	{attribute 'TcIecLibraryType'}
	{attribute 'external_name' := 'F_VN_MultiplyImages_GUID_82AA580E_DA77_541C_61B6_148C085FBCB3'}
	(* Element-wise multiplication of two images using saturation arithmetics. *)
	FUNCTION F_VN_MultiplyImages : HRESULT
	VAR_INPUT
		ipSrcImage1	:	ITcVnImage;	(* First source image *)
		ipSrcImage2	:	ITcVnImage;	(* Second source image *)
		ipDestImage	:	REFERENCE TO ITcVnImage;	(* Destination image (An appropriate destination image will be created if required.) *)
		hrPrev	:	HRESULT;	(* HRESULT indicating the result of previous operations (If SUCCEEDED(hrPrev) equals false, no operation is executed.) *)
	END_VAR

END_FUNCTION

// Functions/Algebraic Image Operations/F_VN_MultiplyImageWithScalar

	{attribute 'TcIecLibraryType'}
	{attribute 'external_name' := 'F_VN_MultiplyImageWithScalar_GUID_B12B22BD_02D6_587A_7D30_3355393075B2'}
	(* Multiply each image pixel by a scalar value using saturation arithmetics. *)
	FUNCTION F_VN_MultiplyImageWithScalar : HRESULT
	VAR_INPUT
		fScalar	:	LREAL;	(* Scalar value *)
		ipSrcImage	:	ITcVnImage;	(* Source image *)
		ipDestImage	:	REFERENCE TO ITcVnImage;	(* Destination image (An appropriate destination image will be created if required.) *)
		hrPrev	:	HRESULT;	(* HRESULT indicating the result of previous operations (If SUCCEEDED(hrPrev) equals false, no operation is executed.) *)
	END_VAR

END_FUNCTION

// Functions/Algebraic Image Operations/F_VN_MultiplyImageWithVector

	{attribute 'TcIecLibraryType'}
	{attribute 'external_name' := 'F_VN_MultiplyImageWithVector_GUID_5A56ACBB_6C80_5F28_4A45_B28BE648BFEA'}
	(* Multiply each image pixel by a vector (1 element for each image channel) using saturation arithmetics. *)
	FUNCTION F_VN_MultiplyImageWithVector : HRESULT
	VAR_INPUT
		aVector	:	REFERENCE TO TcVnVector4_LREAL;	(* 4-element vector (1 element for each image channel. If the image has less channels, the further vector elements are ignored.) *)
		ipSrcImage	:	ITcVnImage;	(* Source image *)
		ipDestImage	:	REFERENCE TO ITcVnImage;	(* Destination image (An appropriate destination image will be created if required.) *)
		hrPrev	:	HRESULT;	(* HRESULT indicating the result of previous operations (If SUCCEEDED(hrPrev) equals false, no operation is executed.) *)
	END_VAR

END_FUNCTION

// Functions/Algebraic Image Operations/F_VN_SubtractImageFromScalar

	{attribute 'TcIecLibraryType'}
	{attribute 'external_name' := 'F_VN_SubtractImageFromScalar_GUID_B8AA2245_74B9_5AC2_4E76_135813C299C9'}
	(* Subtract each image pixel from a scalar value using saturation arithmetics. *)
	FUNCTION F_VN_SubtractImageFromScalar : HRESULT
	VAR_INPUT
		fScalar	:	LREAL;	(* Scalar value *)
		ipSrcImage	:	ITcVnImage;	(* Source image *)
		ipDestImage	:	REFERENCE TO ITcVnImage;	(* Destination image (An appropriate destination image will be created if required.) *)
		hrPrev	:	HRESULT;	(* HRESULT indicating the result of previous operations (If SUCCEEDED(hrPrev) equals false, no operation is executed.) *)
	END_VAR

END_FUNCTION

// Functions/Algebraic Image Operations/F_VN_SubtractImageFromVector

	{attribute 'TcIecLibraryType'}
	{attribute 'external_name' := 'F_VN_SubtractImageFromVector_GUID_17517F7A_96FF_563D_5F02_C474E2D7CC0C'}
	(* Subtract each image pixel from a vector (1 element for each image channel) using saturation arithmetics. *)
	FUNCTION F_VN_SubtractImageFromVector : HRESULT
	VAR_INPUT
		aVector	:	REFERENCE TO TcVnVector4_LREAL;	(* 4-element vector (1 element for each image channel. If the image has less channels, the further vector elements are ignored.) *)
		ipSrcImage	:	ITcVnImage;	(* Source image *)
		ipDestImage	:	REFERENCE TO ITcVnImage;	(* Destination image (An appropriate destination image will be created if required.) *)
		hrPrev	:	HRESULT;	(* HRESULT indicating the result of previous operations (If SUCCEEDED(hrPrev) equals false, no operation is executed.) *)
	END_VAR

END_FUNCTION

// Functions/Algebraic Image Operations/F_VN_SubtractImages

	{attribute 'TcIecLibraryType'}
	{attribute 'external_name' := 'F_VN_SubtractImages_GUID_93AB2995_6F42_52A0_4DD8_5441458B881F'}
	(* Element-wise subtraction of two images using saturation arithmetics. *)
	FUNCTION F_VN_SubtractImages : HRESULT
	VAR_INPUT
		ipSrcImage1	:	ITcVnImage;	(* First source image (minuend) *)
		ipSrcImage2	:	ITcVnImage;	(* Second source image (subtrahend) *)
		ipDestImage	:	REFERENCE TO ITcVnImage;	(* Destination image (An appropriate destination image will be created if required.) *)
		hrPrev	:	HRESULT;	(* HRESULT indicating the result of previous operations (If SUCCEEDED(hrPrev) equals false, no operation is executed.) *)
	END_VAR

END_FUNCTION

// Functions/Algebraic Image Operations/F_VN_SubtractScalarFromImage

	{attribute 'TcIecLibraryType'}
	{attribute 'external_name' := 'F_VN_SubtractScalarFromImage_GUID_4A75C512_59C5_5BEC_5299_C05E617DC6EB'}
	(* Subtract a scalar value from each image pixel using saturation arithmetics. *)
	FUNCTION F_VN_SubtractScalarFromImage : HRESULT
	VAR_INPUT
		ipSrcImage	:	ITcVnImage;	(* Source image *)
		fScalar	:	LREAL;	(* Scalar value *)
		ipDestImage	:	REFERENCE TO ITcVnImage;	(* Destination image (An appropriate destination image will be created if required.) *)
		hrPrev	:	HRESULT;	(* HRESULT indicating the result of previous operations (If SUCCEEDED(hrPrev) equals false, no operation is executed.) *)
	END_VAR

END_FUNCTION

// Functions/Algebraic Image Operations/F_VN_SubtractVectorFromImage

	{attribute 'TcIecLibraryType'}
	{attribute 'external_name' := 'F_VN_SubtractVectorFromImage_GUID_3A450D3E_E7EC_586B_54DB_8372F7AAF290'}
	(* Subtract a vector (1 element for each image channel) from each image pixel using saturation arithmetics. *)
	FUNCTION F_VN_SubtractVectorFromImage : HRESULT
	VAR_INPUT
		ipSrcImage	:	ITcVnImage;	(* Source image *)
		aVector	:	REFERENCE TO TcVnVector4_LREAL;	(* 4-element vector (1 element for each image channel. If the image has less channels, the further vector elements are ignored.) *)
		ipDestImage	:	REFERENCE TO ITcVnImage;	(* Destination image (An appropriate destination image will be created if required.) *)
		hrPrev	:	HRESULT;	(* HRESULT indicating the result of previous operations (If SUCCEEDED(hrPrev) equals false, no operation is executed.) *)
	END_VAR

END_FUNCTION

// Functions/Image Analysis/F_VN_CannyEdgeDetection

	{attribute 'TcIecLibraryType'}
	{attribute 'external_name' := 'F_VN_CannyEdgeDetection_GUID_AD5174D6_E5E1_5D48_5694_BB03C2CA2FDE'}
	(* Find edges using the Canny edge detection algorithm. *)
	FUNCTION F_VN_CannyEdgeDetection : HRESULT
	VAR_INPUT
		ipSrcImage	:	ITcVnImage;	(* Source image (elements of type USINT) *)
		ipDestImage	:	REFERENCE TO ITcVnImage;	(* Destination image (elements of type USINT. An appropriate destination image will be created if required.) *)
		fThresholdLow	:	LREAL;	(* Low threshold *)
		fThresholdHigh	:	LREAL;	(* High threshold *)
		hrPrev	:	HRESULT;	(* HRESULT indicating the result of previous operations (If SUCCEEDED(hrPrev) equals false, no operation is executed.) *)
	END_VAR

END_FUNCTION

// Functions/Image Analysis/F_VN_CannyEdgeDetectionExp

	{attribute 'TcIecLibraryType'}
	{attribute 'external_name' := 'F_VN_CannyEdgeDetectionExp_GUID_6D08A1F4_144F_582E_608D_60E37CF3A2B0'}
	(* Find edges using the Canny edge detection algorithm. (expert function) *)
	FUNCTION F_VN_CannyEdgeDetectionExp : HRESULT
	VAR_INPUT
		ipSrcImage	:	ITcVnImage;	(* Source image (elements of type USINT) *)
		ipDestImage	:	REFERENCE TO ITcVnImage;	(* Destination image (elements of type USINT. An appropriate destination image will be created if required.) *)
		fThresholdLow	:	LREAL;	(* Low threshold *)
		fThresholdHigh	:	LREAL;	(* High threshold *)
		nApertureSize	:	UDINT;	(* Aperture size for the Sobel operator (3, 5, 7) *)
		bL2Gradient	:	BOOL;	(* If true, the more accurate (and slower) L2 norm is used instead of the L1 norm *)
		hrPrev	:	HRESULT;	(* HRESULT indicating the result of previous operations (If SUCCEEDED(hrPrev) equals false, no operation is executed.) *)
	END_VAR

END_FUNCTION

// Functions/Image Analysis/F_VN_CountNonZeroPixels

	{attribute 'TcIecLibraryType'}
	{attribute 'external_name' := 'F_VN_CountNonZeroPixels_GUID_9D27D17F_B34D_59A9_5A50_23FA7CA7A721'}
	(* Counts the non-zero pixels in a single-channel image (e.g. useful to analyze threshold results). *)
	FUNCTION F_VN_CountNonZeroPixels : HRESULT
	VAR_INPUT
		ipSrcImage	:	ITcVnImage;	(* Source image (1 channel) *)
		nNonZero	:	REFERENCE TO ULINT;	(* Returns the number of non-zero pixels in ipSrcImage *)
		hrPrev	:	HRESULT;	(* HRESULT indicating the result of previous operations (If SUCCEEDED(hrPrev) equals false, no operation is executed.) *)
	END_VAR

END_FUNCTION

// Functions/Image Analysis/F_VN_DistanceTransformation

	{attribute 'TcIecLibraryType'}
	{attribute 'external_name' := 'F_VN_DistanceTransformation_GUID_4E9A92BB_223F_5813_612F_9AC3CDD271BA'}
	(* Calculates the distance transformation, which is the distance to the closest zero pixel in a binary image. *)
	FUNCTION F_VN_DistanceTransformation : HRESULT
	VAR_INPUT
		ipSrcImage	:	ITcVnImage;	(* Source image (USINT, 1 channel) *)
		ipDestImage	:	REFERENCE TO ITcVnImage;	(* Destination image (REAL, 1 channel. An appropriate destination image will be created if required.) *)
		eDistanceType	:	ETcVnDistanceType;	(* Distance computation method (supported: L1, L2, C) *)
		eMaskSize	:	ETcVnDistanceTransformationMask;	(* Size of the distance transformation mask *)
		hrPrev	:	HRESULT;	(* HRESULT indicating the result of previous operations (If SUCCEEDED(hrPrev) equals false, no operation is executed.) *)
	END_VAR

END_FUNCTION

// Functions/Image Analysis/F_VN_DistanceTransformationExp

	{attribute 'TcIecLibraryType'}
	{attribute 'external_name' := 'F_VN_DistanceTransformationExp_GUID_4CFD3356_1E5B_593C_50A2_5B385695B3A8'}
	(* Calculates the distance transformation, which is the distance to the closest zero pixel in a binary image. Additionally, an image with component labels is created (discrete Voronoi diagram). (expert function) *)
	FUNCTION F_VN_DistanceTransformationExp : HRESULT
	VAR_INPUT
		ipSrcImage	:	ITcVnImage;	(* Source image (USINT, 1 channel) *)
		ipDestImage	:	REFERENCE TO ITcVnImage;	(* Destination image (REAL, 1 channel. An appropriate destination image will be created if required.) *)
		eDistanceType	:	ETcVnDistanceType;	(* Distance computation method (supported: L1, L2, C) *)
		eMaskSize	:	ETcVnDistanceTransformationMask;	(* Size of the distance transformation mask (PRECISE not supported for label computation) *)
		ipDestLabels	:	REFERENCE TO ITcVnImage;	(* Returns the component labels (Discrete Voronoi diagram; DINT, 1 channel. An appropriate image will be created if required.) *)
		eLabelType	:	ETcVnDistanceTransformationLabel;	(* Type of the labels *)
		hrPrev	:	HRESULT;	(* HRESULT indicating the result of previous operations (If SUCCEEDED(hrPrev) equals false, no operation is executed.) *)
	END_VAR

END_FUNCTION

// Functions/Image Analysis/F_VN_ImageAverage

	{attribute 'TcIecLibraryType'}
	{attribute 'external_name' := 'F_VN_ImageAverage_GUID_0DC2BD23_CB73_5BA1_616F_C8484EB24FBF'}
	(* Computes the (channel-wise) average pixel value of an image. *)
	FUNCTION F_VN_ImageAverage : HRESULT
	VAR_INPUT
		ipSrcImage	:	ITcVnImage;	(* Source image (1 - 4 channels) *)
		aAverage	:	REFERENCE TO TcVnVector4_LREAL;	(* Returns the (channel-wise) average pixel value of ipSrcImage *)
		hrPrev	:	HRESULT;	(* HRESULT indicating the result of previous operations (If SUCCEEDED(hrPrev) equals false, no operation is executed.) *)
	END_VAR

END_FUNCTION

// Functions/Image Analysis/F_VN_ImageAverageExp

	{attribute 'TcIecLibraryType'}
	{attribute 'external_name' := 'F_VN_ImageAverageExp_GUID_CD945797_3224_5304_40E0_D5F68890D6C4'}
	(* Computes the (channel-wise) average pixel value of an image. (expert function) *)
	FUNCTION F_VN_ImageAverageExp : HRESULT
	VAR_INPUT
		ipSrcImage	:	ITcVnImage;	(* Source image (1 - 4 channels) *)
		aAverage	:	REFERENCE TO TcVnVector4_LREAL;	(* Returns the (channel-wise) average pixel value of ipSrcImage *)
		ipMask	:	ITcVnImage;	(* Mask of type USINT (1 channel) *)
		hrPrev	:	HRESULT;	(* HRESULT indicating the result of previous operations (If SUCCEEDED(hrPrev) equals false, no operation is executed.) *)
	END_VAR

END_FUNCTION

// Functions/Image Analysis/F_VN_ImageAverageStdDev

	{attribute 'TcIecLibraryType'}
	{attribute 'external_name' := 'F_VN_ImageAverageStdDev_GUID_3A06BDFA_8386_5D4D_64B1_BCCE83C4268B'}
	(* Computes the (channel-wise) average pixel value and the corresponding standard deviation of an image. *)
	FUNCTION F_VN_ImageAverageStdDev : HRESULT
	VAR_INPUT
		ipSrcImage	:	ITcVnImage;	(* Source image (1 - 4 channels) *)
		aAverage	:	REFERENCE TO TcVnVector4_LREAL;	(* Returns the (channel-wise) average pixel value of ipSrcImage *)
		aStdDev	:	REFERENCE TO TcVnVector4_LREAL;	(* Returns the (channel-wise) pixel value standard deviation of ipSrcImage *)
		hrPrev	:	HRESULT;	(* HRESULT indicating the result of previous operations (If SUCCEEDED(hrPrev) equals false, no operation is executed.) *)
	END_VAR

END_FUNCTION

// Functions/Image Analysis/F_VN_ImageAverageStdDevExp

	{attribute 'TcIecLibraryType'}
	{attribute 'external_name' := 'F_VN_ImageAverageStdDevExp_GUID_752B7A3B_2B8C_5DD8_40E1_0CB9AA5549BC'}
	(* Computes the (channel-wise) average pixel value and the corresponding standard deviation of an image. (expert function) *)
	FUNCTION F_VN_ImageAverageStdDevExp : HRESULT
	VAR_INPUT
		ipSrcImage	:	ITcVnImage;	(* Source image (1 - 4 channels) *)
		aAverage	:	REFERENCE TO TcVnVector4_LREAL;	(* Returns the (channel-wise) average pixel value of ipSrcImage *)
		aStdDev	:	REFERENCE TO TcVnVector4_LREAL;	(* Returns the (channel-wise) pixel value standard deviation of ipSrcImage *)
		ipMask	:	ITcVnImage;	(* Mask of type USINT (1 channel) *)
		hrPrev	:	HRESULT;	(* HRESULT indicating the result of previous operations (If SUCCEEDED(hrPrev) equals false, no operation is executed.) *)
	END_VAR

END_FUNCTION

// Functions/Image Analysis/F_VN_ImageCenterOfMass

	{attribute 'TcIecLibraryType'}
	{attribute 'external_name' := 'F_VN_ImageCenterOfMass_GUID_11DF4D3B_5664_5D62_5346_5D36F2E2BFDE'}
	(* Computes the center of mass of an image. *)
	FUNCTION F_VN_ImageCenterOfMass : HRESULT
	VAR_INPUT
		ipSrcImage	:	ITcVnImage;	(* Source image *)
		aCenterOfMass	:	REFERENCE TO TcVnPoint2_LREAL;	(* Returns the center of mass of the image *)
		hrPrev	:	HRESULT;	(* HRESULT indicating the result of previous operations (If SUCCEEDED(hrPrev) equals false, no operation is executed.) *)
	END_VAR

END_FUNCTION

// Functions/Image Analysis/F_VN_ImageCenterOfMassExp

	{attribute 'TcIecLibraryType'}
	{attribute 'external_name' := 'F_VN_ImageCenterOfMassExp_GUID_AA5EE9CE_0D3F_5D4D_4151_3F6E4694BA31'}
	(* Computes the center of mass of an image. *)
	FUNCTION F_VN_ImageCenterOfMassExp : HRESULT
	VAR_INPUT
		ipSrcImage	:	ITcVnImage;	(* Source image *)
		aCenterOfMass	:	REFERENCE TO TcVnPoint2_LREAL;	(* Returns the center of mass of the image *)
		ipMask	:	ITcVnImage;	(* Mask of type USINT *)
		hrPrev	:	HRESULT;	(* HRESULT indicating the result of previous operations (If SUCCEEDED(hrPrev) equals false, no operation is executed.) *)
	END_VAR

END_FUNCTION

// Functions/Image Analysis/F_VN_ImageMedian

	{attribute 'TcIecLibraryType'}
	{attribute 'external_name' := 'F_VN_ImageMedian_GUID_0749BAFE_9F4A_5160_6F6A_8AABC6BC5ADF'}
	(* Computes the (approximated, channel-wise) median pixel value of an image. *)
	FUNCTION F_VN_ImageMedian : HRESULT
	VAR_INPUT
		ipSrcImage	:	ITcVnImage;	(* Source image (1 - 4 channels) *)
		aMedian	:	REFERENCE TO TcVnVector4_LREAL;	(* Returns the (approximated, channel-wise) median pixel value of ipSrcImage *)
		hrPrev	:	HRESULT;	(* HRESULT indicating the result of previous operations (If SUCCEEDED(hrPrev) equals false, no operation is executed.) *)
	END_VAR

END_FUNCTION

// Functions/Image Analysis/F_VN_ImageMedianExp

	{attribute 'TcIecLibraryType'}
	{attribute 'external_name' := 'F_VN_ImageMedianExp_GUID_878FED6A_584C_5450_4696_A375FCEC6A14'}
	(* Computes the (approximated, channel-wise) median pixel value of an image. (expert function) *)
	FUNCTION F_VN_ImageMedianExp : HRESULT
	VAR_INPUT
		ipSrcImage	:	ITcVnImage;	(* Source image (1 - 4 channels) *)
		aMedian	:	REFERENCE TO TcVnVector4_LREAL;	(* Returns the (approximated, channel-wise) median pixel value of ipSrcImage *)
		ipMask	:	ITcVnImage;	(* Mask of type USINT (1 channel) *)
		hrPrev	:	HRESULT;	(* HRESULT indicating the result of previous operations (If SUCCEEDED(hrPrev) equals false, no operation is executed.) *)
	END_VAR

END_FUNCTION

// Functions/Image Analysis/F_VN_ImageMoments

	{attribute 'TcIecLibraryType'}
	{attribute 'external_name' := 'F_VN_ImageMoments_GUID_15556A38_7F53_5846_64D1_5689BA19D98B'}
	(* Computes the spatial moments, the central moments, and the central normalized moments of an image up to the third order. *)
	FUNCTION F_VN_ImageMoments : HRESULT
	VAR_INPUT
		ipImage	:	ITcVnImage;	(* Source image (1 channel, elements of type USINT or REAL) *)
		stMoments	:	REFERENCE TO TcVnMoments;	(* Returns a struct containing the moments *)
		bBinaryImage	:	BOOL;	(* If true, all non-zero pixels are treated as ones *)
		hrPrev	:	HRESULT;	(* HRESULT indicating the result of previous operations (If SUCCEEDED(hrPrev) equals false, no operation is executed.) *)
	END_VAR

END_FUNCTION

// Functions/Image Analysis/F_VN_MaxPixelValue

	{attribute 'TcIecLibraryType'}
	{attribute 'external_name' := 'F_VN_MaxPixelValue_GUID_C2109E0C_B3DB_59C6_566D_9F2FA6754D3B'}
	(* Finds the maximum pixel value in an image (1 - 4 channels supported). *)
	FUNCTION F_VN_MaxPixelValue : HRESULT
	VAR_INPUT
		ipImage	:	ITcVnImage;	(* Source image *)
		aMaxValue	:	REFERENCE TO TcVnVector4_LREAL;	(* Returns the maximum pixel value *)
		aPosition	:	REFERENCE TO TcVnPoint2_DINT;	(* Returns the first found position of aMaxValue *)
		hrPrev	:	HRESULT;	(* HRESULT indicating the result of previous operations (If SUCCEEDED(hrPrev) equals false, no operation is executed.) *)
	END_VAR

END_FUNCTION

// Functions/Image Analysis/F_VN_MaxPixelValueExp

	{attribute 'TcIecLibraryType'}
	{attribute 'external_name' := 'F_VN_MaxPixelValueExp_GUID_EECB76E7_3726_5026_5DAD_97DC6E3892F6'}
	(* Finds the maximum pixel value in an image (1 - 4 channels supported). (expert function) *)
	FUNCTION F_VN_MaxPixelValueExp : HRESULT
	VAR_INPUT
		ipImage	:	ITcVnImage;	(* Source image *)
		aMaxValue	:	REFERENCE TO TcVnVector4_LREAL;	(* Returns the maximum pixel value *)
		aPosition	:	REFERENCE TO TcVnPoint2_DINT;	(* Returns the first found position of aMaxValue (not supported for multi-channel images with ELEMENTWISE) *)
		ipMask	:	ITcVnImage;	(* Optional mask to specify which pixel positions are considered (USINT, set parameter to 0 if not required) *)
		eVectorCompareMethod	:	ETcVnVectorCompareMethod;	(* Select a vector compare method for multi-channel images *)
		hrPrev	:	HRESULT;	(* HRESULT indicating the result of previous operations (If SUCCEEDED(hrPrev) equals false, no operation is executed.) *)
	END_VAR

END_FUNCTION

// Functions/Image Analysis/F_VN_MinPixelValue

	{attribute 'TcIecLibraryType'}
	{attribute 'external_name' := 'F_VN_MinPixelValue_GUID_AFFC0405_606C_50EB_719C_80B83B579EAE'}
	(* Finds the minimum pixel value in an image (1 - 4 channels supported). *)
	FUNCTION F_VN_MinPixelValue : HRESULT
	VAR_INPUT
		ipImage	:	ITcVnImage;	(* Source image *)
		aMinValue	:	REFERENCE TO TcVnVector4_LREAL;	(* Returns the minimum pixel value *)
		aPosition	:	REFERENCE TO TcVnPoint2_DINT;	(* Returns the first found position of aMinValue *)
		hrPrev	:	HRESULT;	(* HRESULT indicating the result of previous operations (If SUCCEEDED(hrPrev) equals false, no operation is executed.) *)
	END_VAR

END_FUNCTION

// Functions/Image Analysis/F_VN_MinPixelValueExp

	{attribute 'TcIecLibraryType'}
	{attribute 'external_name' := 'F_VN_MinPixelValueExp_GUID_778ECF13_218D_51F8_450E_7F6CA400858A'}
	(* Finds the minimum pixel value in an image (1 - 4 channels supported). (expert function) *)
	FUNCTION F_VN_MinPixelValueExp : HRESULT
	VAR_INPUT
		ipImage	:	ITcVnImage;	(* Source image *)
		aMinValue	:	REFERENCE TO TcVnVector4_LREAL;	(* Returns the minimum pixel value *)
		aPosition	:	REFERENCE TO TcVnPoint2_DINT;	(* Returns the first found position of aMinValue (not supported for multi-channel images with ELEMENTWISE) *)
		ipMask	:	ITcVnImage;	(* Optional mask to specify which pixel positions are considered (USINT, set parameter to 0 if not required) *)
		eVectorCompareMethod	:	ETcVnVectorCompareMethod;	(* Select a vector compare method for multi-channel images *)
		hrPrev	:	HRESULT;	(* HRESULT indicating the result of previous operations (If SUCCEEDED(hrPrev) equals false, no operation is executed.) *)
	END_VAR

END_FUNCTION

// Functions/Measurement/F_VN_AdjustSearchWindowOrientationToLinearEdge

	{attribute 'TcIecLibraryType'}
	{attribute 'external_name' := 'F_VN_AdjustSearchWindowOrientationToLinearEdge_GUID_27A0ECAC_187C_5D0A_69E7_C784A5DCE9CD'}
	(* Adjust the search window to be orthogonal to a linear edge. Might be helpful before calling edge localization and distance measurement functions that rely on the search window. *)
	FUNCTION F_VN_AdjustSearchWindowOrientationToLinearEdge : HRESULT
	VAR_INPUT
		ipSrcImage	:	ITcVnImage;	(* Source image *)
		aStartPoint	:	REFERENCE TO TcVnPoint2_REAL;	(* Position from which to start the search process (in the direction of aEndPoint), which is not changed *)
		aEndPoint	:	REFERENCE TO TcVnPoint2_REAL;	(* Position where the search process ends, which is adjusted by this function *)
		eEdgeDirection	:	ETcVnEdgeDirection;	(* Specification of the edge direction to search for *)
		fMinStrength	:	REAL;	(* Specification of the minimum strength (intensity difference) of the edge to search for *)
		nMaxThickness	:	UDINT;	(* Specification of the maximum thickness of the edge to search for, which means fMinStrength must be reached within nMaxThickness pixels *)
		nSearchLines	:	UDINT;	(* Width of the search window, i.e. the number of search lines (3, 5, 7, ...), centered around the line specified by aStartPoint and aEndPoint *)
		hrPrev	:	HRESULT;	(* HRESULT indicating the result of previous operations (If SUCCEEDED(hrPrev) equals false, no operation is executed.) *)
	END_VAR

END_FUNCTION

// Functions/Measurement/F_VN_ClosestPointsBF

	{attribute 'TcIecLibraryType'}
	{attribute 'external_name' := 'F_VN_ClosestPointsBF_GUID_942CB598_7FEE_5119_5542_9CC86CD424CE'}
	(* Find the closest distance between two 2d point sets of the same type, using a brute force approach. *)
	FUNCTION F_VN_ClosestPointsBF : HRESULT
	VAR_INPUT
		ipPointSet1	:	ITcVnContainer;	(* Container with 1st set of 2d points *)
		ipPointSet2	:	ITcVnContainer;	(* Container with 2nd set of 2d points *)
		fMinDist	:	REFERENCE TO LREAL;	(* Returns the minimum distance between 2 points of the different point sets *)
		aPoint1	:	REFERENCE TO TcVnPoint2_LREAL;	(* Returns the point out of ipPointSet1, for which fMinDist is achieved *)
		aPoint2	:	REFERENCE TO TcVnPoint2_LREAL;	(* Returns the point out of ipPointSet2, for which fMinDist is achieved *)
		hrPrev	:	HRESULT;	(* HRESULT indicating the result of previous operations (If SUCCEEDED(hrPrev) equals false, no operation is executed.) *)
	END_VAR

END_FUNCTION

// Functions/Measurement/F_VN_LocateCircularArc

	{attribute 'TcIecLibraryType'}
	{attribute 'external_name' := 'F_VN_LocateCircularArc_GUID_30C14ED2_0EBE_5080_6499_B7B697FA6815'}
	(* Locate a circular arc, using an interpolation method. *)
	FUNCTION F_VN_LocateCircularArc : HRESULT
	VAR_INPUT
		ipSrcImage	:	ITcVnImage;	(* Source image (1 channel) *)
		stCircularArc	:	REFERENCE TO TcVnCircularArc;	(* Returns the circular arc parameters *)
		aCenter	:	REFERENCE TO TcVnPoint2_REAL;	(* Input estimated circle center (only used as a starting point to search for the circle contour, not used for the circle center estimation) *)
		fSearchRadius	:	REAL;	(* Input search radius (starting from aCenter, should be greater than the actual circle radius but aCenter + fSearchRadius should be within the image borders) *)
		fArcDirectionRad	:	LREAL;	(* Input search starting direction in radian. Valid range is [-pi, +pi], where right is 0 rad, top is -pi/2 rad and bottom +pi/2 rad. The circular arc should at least be valid in range fArcDirectionRad +- 0.4 rad. *)
		eEdgeDirection	:	ETcVnEdgeDirection;	(* Specification of the edge direction to search for *)
		fMinStrength	:	REAL;	(* Specification of the minimum strength (intensity difference) of the edge to search for *)
		hrPrev	:	HRESULT;	(* HRESULT indicating the result of previous operations (If SUCCEEDED(hrPrev) equals false, no operation is executed.) *)
	END_VAR

END_FUNCTION

// Functions/Measurement/F_VN_LocateCircularArcExp

	{attribute 'TcIecLibraryType'}
	{attribute 'external_name' := 'F_VN_LocateCircularArcExp_GUID_BECFD49B_4206_5CF0_51A9_EB8B13BA786C'}
	(* Locate a circular arc. (expert function) *)
	FUNCTION F_VN_LocateCircularArcExp : HRESULT
	VAR_INPUT
		ipSrcImage	:	ITcVnImage;	(* Source image (1 channel) *)
		stCircularArc	:	REFERENCE TO TcVnCircularArc;	(* Returns the circular arc parameters *)
		aCenter	:	REFERENCE TO TcVnPoint2_REAL;	(* Input estimated circle center (only used as a starting point to search for the circle contour, not used for the circle center estimation) *)
		fSearchRadius	:	REAL;	(* Input search radius (starting from aCenter, should be greater than the actual circle radius but aCenter + fSearchRadius should be within the image borders) *)
		fArcDirectionRad	:	LREAL;	(* Input search starting direction in radian. Valid range is [-pi, +pi], where right is 0 rad, top is -pi/2 rad and bottom +pi/2 rad. The circular arc should at least be valid in range fArcDirectionRad +- 4 * fAngleStepRad) *)
		eEdgeDirection	:	ETcVnEdgeDirection;	(* Specification of the edge direction to search for *)
		fMinStrength	:	REAL;	(* Specification of the minimum strength (intensity difference) of the edge to search for *)
		fAngleStepRad	:	LREAL;	(* Search step in rad (should be chosen so that about 20 - 60 steps are available for the whole arc. In most cases 0.1 rad (5.7 deg) is a good value) *)
		nMaxThickness	:	UDINT;	(* Specification of the maximum thickness of the edge to search for, which means fMinStrength must be reached within nMaxThickness pixels *)
		bInvertSearchDirection	:	BOOL;	(* If true, the search starts from outside the circular arc in direction of the center *)
		nSubpixelsIterations	:	UDINT;	(* Specifies the number of subpixels (for INTERPOLATION, 10 - 20 usually is sufficient) or maximum number of iterations for optimizing the parameters (for APPROX_ERF and APPROX_GAUSSIAN, 100 usually is sufficient) *)
		fApproxPrecision	:	REAL;	(* Specifies the approximation precision for APPROX_ERF and APPROX_GAUSSIAN (0.0001 usually is sufficient, unused for INTERPOLATION) *)
		eAlgorithm	:	ETcVnEdgeDetectionAlgorithm;	(* Selection of the edge detection algorithm *)
		ipContourPoints	:	REFERENCE TO ITcVnContainer;	(* Returns the subpixel accurate contour (optional, set to 0 if not required; ContainerType_Vector_TcVnPoint2_REAL; Non-zero interface pointers are reused.) *)
		hrPrev	:	HRESULT;	(* HRESULT indicating the result of previous operations (If SUCCEEDED(hrPrev) equals false, no operation is executed.) *)
	END_VAR

END_FUNCTION

// Functions/Measurement/F_VN_LocateEdge

	{attribute 'TcIecLibraryType'}
	{attribute 'external_name' := 'F_VN_LocateEdge_GUID_013D6F07_158B_5F4E_4B22_5957300955E9'}
	(* Locate the points of the first occuring edge inside a specified search window, using an interpolation method. *)
	FUNCTION F_VN_LocateEdge : HRESULT
	VAR_INPUT
		ipSrcImage	:	ITcVnImage;	(* Source image (1 channel) *)
		ipEdgePoints	:	REFERENCE TO ITcVnContainer;	(* Returns the detected edge points (ContainerType_Vector_TcVnPoint2_REAL) *)
		aStartPoint	:	REFERENCE TO TcVnPoint2_REAL;	(* Position from which to start the search process (in the direction of aEndPoint) *)
		aEndPoint	:	REFERENCE TO TcVnPoint2_REAL;	(* Position where the search process ends *)
		eEdgeDirection	:	ETcVnEdgeDirection;	(* Specification of the edge direction to search for *)
		fMinStrength	:	REAL;	(* Specification of the minimum strength (intensity difference) of the edge to search for *)
		nSearchLines	:	UDINT;	(* Width of the search window, i.e. the number of search lines (1, 3, 5, 7, ...), centered around the line specified by aStartPoint and aEndPoint *)
		hrPrev	:	HRESULT;	(* HRESULT indicating the result of previous operations (If SUCCEEDED(hrPrev) equals false, no operation is executed.) *)
	END_VAR
	VAR_OUTPUT
		fAvgStrength	:	REAL;	(* Returns the average strength of the detected edge *)
	END_VAR

END_FUNCTION

// Functions/Measurement/F_VN_LocateEdgeExp

	{attribute 'TcIecLibraryType'}
	{attribute 'external_name' := 'F_VN_LocateEdgeExp_GUID_1DDE9ACC_6084_5FBA_7F3B_01F41DA4B4EC'}
	(* Locate the points of the first occuring edge inside a specified search window with subpixel accuracy. (expert function) *)
	FUNCTION F_VN_LocateEdgeExp : HRESULT
	VAR_INPUT
		ipSrcImage	:	ITcVnImage;	(* Source image (1 channel) *)
		ipEdgePoints	:	REFERENCE TO ITcVnContainer;	(* Returns the detected edge points (ContainerType_Vector_TcVnPoint2_REAL) *)
		aStartPoint	:	REFERENCE TO TcVnPoint2_REAL;	(* Position from which to start the search process (in the direction of aEndPoint) *)
		aEndPoint	:	REFERENCE TO TcVnPoint2_REAL;	(* Position where the search process ends *)
		eEdgeDirection	:	ETcVnEdgeDirection;	(* Specification of the edge direction to search for *)
		fMinStrength	:	REAL;	(* Specification of the minimum strength (intensity difference) of the edge to search for *)
		nSearchLines	:	UDINT;	(* Width of the search window, i.e. the number of search lines (1, 3, 5, 7, ...), centered around the line specified by aStartPoint and aEndPoint *)
		fSearchLineDist	:	REAL;	(* Distance between the search lines in pixels (> 0) *)
		nMaxThickness	:	UDINT;	(* Specification of the maximum thickness of the edge to search for, which means fMinStrength must be reached within nMaxThickness pixels *)
		nSubpixelsIterations	:	UDINT;	(* Specifies the number of subpixels (for INTERPOLATION, 10 - 20 usually is sufficient) or maximum number of iterations for optimizing the parameters (for APPROX_ERF and APPROX_GAUSSIAN, 100 usually is sufficient) *)
		fApproxPrecision	:	REAL;	(* Specifies the approximation precision for APPROX_ERF and APPROX_GAUSSIAN (0.0001 usually is sufficient, unused for INTERPOLATION) *)
		eAlgorithm	:	ETcVnEdgeDetectionAlgorithm;	(* Selection of the edge detection algorithm *)
		hrPrev	:	HRESULT;	(* HRESULT indicating the result of previous operations (If SUCCEEDED(hrPrev) equals false, no operation is executed.) *)
	END_VAR
	VAR_OUTPUT
		fAvgStrength	:	REAL;	(* Returns the average strength of the detected edge *)
	END_VAR

END_FUNCTION

// Functions/Measurement/F_VN_LocateEdges

	{attribute 'TcIecLibraryType'}
	{attribute 'external_name' := 'F_VN_LocateEdges_GUID_7A95BAA9_7AF5_58BB_412E_BC269953AF81'}
	(* Locate the points of multiple occuring edges inside a specified search window, using an interpolation method. *)
	FUNCTION F_VN_LocateEdges : HRESULT
	VAR_INPUT
		ipSrcImage	:	ITcVnImage;	(* Source image (1 channel) *)
		ipEdgePoints	:	REFERENCE TO ITcVnContainer;	(* Returns the detected edge points (ContainerType_Vector_Vector_TcVnPoint2_REAL) *)
		aStartPoint	:	REFERENCE TO TcVnPoint2_REAL;	(* Position from which to start the search process (in the direction of aEndPoint) *)
		aEndPoint	:	REFERENCE TO TcVnPoint2_REAL;	(* Position where the search process ends *)
		nNumEdges	:	UDINT;	(* The (maximum) number of edges to search for *)
		eEdgeDirection	:	ETcVnEdgeDirection;	(* Specification of the edge direction to search for *)
		bAlternateDirection	:	BOOL;	(* If true, eEdgeDirection is alternated after each detected edge. Else, only edges with eEdgeDirection are searched for. *)
		fMinStrength	:	REAL;	(* Specification of the minimum strength (intensity difference) of the edge to search for *)
		nSearchLines	:	UDINT;	(* Width of the search window, i.e. the number of search lines (1, 3, 5, 7, ...), centered around the line specified by aStartPoint and aEndPoint *)
		hrPrev	:	HRESULT;	(* HRESULT indicating the result of previous operations (If SUCCEEDED(hrPrev) equals false, no operation is executed.) *)
	END_VAR
	VAR_OUTPUT
		fAvgStrength	:	REAL;	(* Returns the average strength of the detected edges *)
	END_VAR

END_FUNCTION

// Functions/Measurement/F_VN_LocateEdgesExp

	{attribute 'TcIecLibraryType'}
	{attribute 'external_name' := 'F_VN_LocateEdgesExp_GUID_48F3F565_C08A_5F76_7BD8_6A67CBC1CE6C'}
	(* Locate the points of multiple occuring edges inside a specified search window with subpixel accuracy. (expert function) *)
	FUNCTION F_VN_LocateEdgesExp : HRESULT
	VAR_INPUT
		ipSrcImage	:	ITcVnImage;	(* Source image (1 channel) *)
		ipEdgePoints	:	REFERENCE TO ITcVnContainer;	(* Returns the detected edge points (ContainerType_Vector_Vector_TcVnPoint2_REAL) *)
		aStartPoint	:	REFERENCE TO TcVnPoint2_REAL;	(* Position from which to start the search process (in the direction of aEndPoint) *)
		aEndPoint	:	REFERENCE TO TcVnPoint2_REAL;	(* Position where the search process ends *)
		nNumEdges	:	UDINT;	(* The (maximum) number of edges to search for *)
		eEdgeDirection	:	ETcVnEdgeDirection;	(* Specification of the edge direction to search for *)
		bAlternateDirection	:	BOOL;	(* If true, eEdgeDirection is alternated after each detected edge. Else, only edges with eEdgeDirection are searched for. *)
		fMinStrength	:	REAL;	(* Specification of the minimum strength (intensity difference) of the edge to search for *)
		nSearchLines	:	UDINT;	(* Width of the search window, i.e. the number of search lines (1, 3, 5, 7, ...), centered around the line specified by aStartPoint and aEndPoint *)
		fSearchLineDist	:	REAL;	(* Distance between the search lines in pixels (> 0) *)
		nMaxThickness	:	UDINT;	(* Specification of the maximum thickness of the edge to search for, which means fMinStrength must be reached within nMaxThickness pixels *)
		nSubpixelsIterations	:	UDINT;	(* Specifies the number of subpixels (for INTERPOLATION, 10 - 20 usually is sufficient) or maximum number of iterations for optimizing the parameters (for APPROX_ERF and APPROX_GAUSSIAN, 100 usually is sufficient) *)
		fApproxPrecision	:	REAL;	(* Specifies the approximation precision for APPROX_ERF and APPROX_GAUSSIAN (0.0001 usually is sufficient, unused for INTERPOLATION) *)
		eAlgorithm	:	ETcVnEdgeDetectionAlgorithm;	(* Selection of the edge detection algorithm *)
		hrPrev	:	HRESULT;	(* HRESULT indicating the result of previous operations (If SUCCEEDED(hrPrev) equals false, no operation is executed.) *)
	END_VAR
	VAR_OUTPUT
		fAvgStrength	:	REAL;	(* Returns the average strength of the detected edges *)
	END_VAR

END_FUNCTION

// Functions/Measurement/F_VN_LocateEllipse

	{attribute 'TcIecLibraryType'}
	{attribute 'external_name' := 'F_VN_LocateEllipse_GUID_110B1BB4_407A_5974_7206_63B3CC61A6CE'}
	(* Locate an ellipse, using an interpolation method for locating the edges. *)
	FUNCTION F_VN_LocateEllipse : HRESULT
	VAR_INPUT
		ipSrcImage	:	ITcVnImage;	(* Source image (1 channel) *)
		stEllipse	:	REFERENCE TO TcVnRotatedRectangle;	(* Returns the detected ellipse *)
		aCenter	:	REFERENCE TO TcVnPoint2_REAL;	(* The expected ellipse center *)
		fSearchRadius	:	REAL;	(* Radius around aCenter to search for edges (aCenter + fSearchRadius in all directions must be inside image borders!) *)
		eEdgeDirection	:	ETcVnEdgeDirection;	(* Specification of the edge direction to search for (from center to outside ellipse) *)
		fMinStrength	:	REAL;	(* Specification of the minimum strength (intensity difference) of the edge to search for *)
		hrPrev	:	HRESULT;	(* HRESULT indicating the result of previous operations (If SUCCEEDED(hrPrev) equals false, no operation is executed.) *)
	END_VAR

END_FUNCTION

// Functions/Measurement/F_VN_LocateEllipseExp

	{attribute 'TcIecLibraryType'}
	{attribute 'external_name' := 'F_VN_LocateEllipseExp_GUID_66385D36_3C7B_561F_6FA6_CED763C24A9D'}
	(* Locate an ellipse. (expert function) *)
	FUNCTION F_VN_LocateEllipseExp : HRESULT
	VAR_INPUT
		ipSrcImage	:	ITcVnImage;	(* Source image (1 channel) *)
		stEllipse	:	REFERENCE TO TcVnRotatedRectangle;	(* Returns the detected ellipse *)
		aCenter	:	REFERENCE TO TcVnPoint2_REAL;	(* The expected ellipse center *)
		fSearchRadius	:	REAL;	(* Radius around aCenter to search for edges *)
		eEdgeDirection	:	ETcVnEdgeDirection;	(* Specification of the edge direction to search for (from center to outside ellipse or other way round, if bInvertSearchDirection is true) *)
		fMinStrength	:	REAL;	(* Specification of the minimum strength (intensity difference) of the edge to search for *)
		nMaxThickness	:	UDINT;	(* Specification of the maximum thickness of the edge to search for, which means fMinStrength must be reached within nMaxThickness pixels *)
		bInvertSearchDirection	:	BOOL;	(* If true, the search starts from outside the ellipse in direction of the center *)
		fMinSearchRadius	:	REAL;	(* Radius around aCenter to skip before starting to search for edges (e.g. to save time or if the center contains edges that should be ignored) *)
		nSubpixelsIterations	:	UDINT;	(* Specifies the number of subpixels (for INTERPOLATION, 10 - 20 usually is sufficient) or maximum number of iterations for optimizing the parameters (for APPROX_ERF and APPROX_GAUSSIAN, 100 usually is sufficient) *)
		nSearchLines	:	UDINT;	(* Specifies the amount of search lines, which are equally distributed in all directions (must be >= 8 and a multiple of 4) *)
		fApproxPrecision	:	REAL;	(* Specifies the approximation precision for APPROX_ERF and APPROX_GAUSSIAN (0.0001 usually is sufficient, unused for INTERPOLATION) *)
		eAlgorithm	:	ETcVnEdgeDetectionAlgorithm;	(* Selection of the edge detection algorithm *)
		ipContourPoints	:	REFERENCE TO ITcVnContainer;	(* Returns the subpixel accurate ellipse contour (optional, set to 0 if not required; ContainerType_Vector_TcVnPoint2_REAL; Non-zero interface pointers are reused.) *)
		hrPrev	:	HRESULT;	(* HRESULT indicating the result of previous operations (If SUCCEEDED(hrPrev) equals false, no operation is executed.) *)
	END_VAR

END_FUNCTION

// Functions/Measurement/F_VN_MeasureAngleBetweenEdges

	{attribute 'TcIecLibraryType'}
	{attribute 'external_name' := 'F_VN_MeasureAngleBetweenEdges_GUID_BC1D484F_B613_55A6_6286_1945AA9FD3E5'}
	(* Measure the angle between 2 edges, using an interpolation method. *)
	FUNCTION F_VN_MeasureAngleBetweenEdges : HRESULT
	VAR_INPUT
		ipSrcImage	:	ITcVnImage;	(* Source image (1 channel) *)
		fAngle	:	REFERENCE TO REAL;	(* Returns the angle between the detected edges (radians) *)
		aInnerPoint	:	REFERENCE TO TcVnPoint2_REAL;	(* Position inside the angle to measure, from which to start the edge search process (in the direction of aOuterPoint1 and aOuterPoint2) *)
		aOuterPoint1	:	REFERENCE TO TcVnPoint2_REAL;	(* Position where the search process for edge 1 ends *)
		aOuterPoint2	:	REFERENCE TO TcVnPoint2_REAL;	(* Position where the search process for edge 2 ends *)
		eEdgeDirection	:	ETcVnEdgeDirection;	(* Specification of the edge direction from aInnerPoint to aOuterPoint1 and aOuterPoint2 to search for *)
		fMinStrength	:	REAL;	(* Specification of the minimum strength (intensity difference) of the edge to search for *)
		nSearchLines	:	UDINT;	(* Width of the search windows, i.e. the number of search lines (3, 5, 7, ...), centered around the lines specified by aInnerPoint and aOuterPoint1, aOuterPoint2 *)
		hrPrev	:	HRESULT;	(* HRESULT indicating the result of previous operations (If SUCCEEDED(hrPrev) equals false, no operation is executed.) *)
	END_VAR

END_FUNCTION

// Functions/Measurement/F_VN_MeasureAngleBetweenEdgesExp

	{attribute 'TcIecLibraryType'}
	{attribute 'external_name' := 'F_VN_MeasureAngleBetweenEdgesExp_GUID_D5A463BE_58FE_56F9_549C_DDD60A910254'}
	(* Measure the angle between 2 edges. *)
	FUNCTION F_VN_MeasureAngleBetweenEdgesExp : HRESULT
	VAR_INPUT
		ipSrcImage	:	ITcVnImage;	(* Source image (1 channel) *)
		fAngle	:	REFERENCE TO REAL;	(* Returns the angle between the detected edges (radians or degrees, depending on bAngleInDegrees) *)
		aInnerPoint	:	REFERENCE TO TcVnPoint2_REAL;	(* Position inside the angle to measure, from which to start the edge search process (in the direction of aOuterPoint1 and aOuterPoint2) *)
		aOuterPoint1	:	REFERENCE TO TcVnPoint2_REAL;	(* Position where the search process for edge 1 ends *)
		aOuterPoint2	:	REFERENCE TO TcVnPoint2_REAL;	(* Position where the search process for edge 2 ends *)
		eEdgeDirection	:	ETcVnEdgeDirection;	(* Specification of the edge direction from aInnerPoint to aOuterPoint1 and aOuterPoint2 to search for *)
		fMinStrength	:	REAL;	(* Specification of the minimum strength (intensity difference) of the edge to search for *)
		nSearchLines	:	UDINT;	(* Width of the search window, i.e. the number of search lines (3, 5, 7, ...), centered around the line specified by aInnerPoint and aOuterPoint1, aOuterPoint2 *)
		fSearchLineDist	:	REAL;	(* Distance between the search lines in pixels (> 0) *)
		nMaxThickness	:	UDINT;	(* Specification of the maximum thickness of the edge to search for, which means fMinStrength must be reached within nMaxThickness pixels *)
		bInvertSearchDirection	:	BOOL;	(* If true, the search starts from each aOuterPoint in direction of aInnerPoint *)
		nSubpixelsIterations	:	UDINT;	(* Specifies the number of subpixels (for INTERPOLATION, 10 - 20 usually is sufficient) or maximum number of iterations for optimizing the parameters (for APPROX_ERF and APPROX_GAUSSIAN, 100 usually is sufficient) *)
		bAngleInDegrees	:	BOOL;	(* fAngle is in degrees, if true *)
		fApproxPrecision	:	REAL;	(* Specifies the approximation precision for APPROX_ERF and APPROX_GAUSSIAN (0.0001 usually is sufficient, unused for INTERPOLATION) *)
		eAlgorithm	:	ETcVnEdgeDetectionAlgorithm;	(* Selection of the edge detection algorithm *)
		ipEdgePoints1	:	REFERENCE TO ITcVnContainer;	(* Returns the detected edge points between aInnerPoint and aOuterPoint1 (ContainerType_Vector_TcVnPoint2_REAL) *)
		ipEdgePoints2	:	REFERENCE TO ITcVnContainer;	(* Returns the detected edge points between aInnerPoint and aOuterPoint2 (ContainerType_Vector_TcVnPoint2_REAL) *)
		hrPrev	:	HRESULT;	(* HRESULT indicating the result of previous operations (If SUCCEEDED(hrPrev) equals false, no operation is executed.) *)
	END_VAR

END_FUNCTION

// Functions/Measurement/F_VN_MeasureEdgeDistance

	{attribute 'TcIecLibraryType'}
	{attribute 'external_name' := 'F_VN_MeasureEdgeDistance_GUID_0769A961_12AF_5CB1_6944_95791D3EBED0'}
	(* Measure the distance between 2 parallel edges, using an interpolation method. *)
	FUNCTION F_VN_MeasureEdgeDistance : HRESULT
	VAR_INPUT
		ipSrcImage	:	ITcVnImage;	(* Source image (1 channel) *)
		fAvgDistance	:	REFERENCE TO REAL;	(* Returns the average distance between the detected edges *)
		aStartPoint	:	REFERENCE TO TcVnPoint2_REAL;	(* Position from which to start the search process (in the direction of aEndPoint) *)
		aEndPoint	:	REFERENCE TO TcVnPoint2_REAL;	(* Position where the search process ends *)
		eEdgeDirection	:	ETcVnEdgeDirection;	(* Specification of the edge direction from aStartPoint to aEndPoint to search for *)
		fMinStrength	:	REAL;	(* Specification of the minimum strength (intensity difference) of the edge to search for *)
		nSearchLines	:	UDINT;	(* Width of the search window, i.e. the number of search lines (1, 3, 5, 7, ...), centered around the line specified by aStartPoint and aEndPoint *)
		hrPrev	:	HRESULT;	(* HRESULT indicating the result of previous operations (If SUCCEEDED(hrPrev) equals false, no operation is executed.) *)
	END_VAR

END_FUNCTION

// Functions/Measurement/F_VN_MeasureEdgeDistanceExp

	{attribute 'TcIecLibraryType'}
	{attribute 'external_name' := 'F_VN_MeasureEdgeDistanceExp_GUID_D9FE7A5B_9C38_521B_6575_D524EABA6B69'}
	(* Measure the distance between 2 parallel edges. (expert function) *)
	FUNCTION F_VN_MeasureEdgeDistanceExp : HRESULT
	VAR_INPUT
		ipSrcImage	:	ITcVnImage;	(* Source image (1 channel) *)
		fAvgDistance	:	REFERENCE TO REAL;	(* Returns the average distance between the detected edges *)
		aStartPoint	:	REFERENCE TO TcVnPoint2_REAL;	(* Position from which to start the search process (in the direction of aEndPoint) *)
		aEndPoint	:	REFERENCE TO TcVnPoint2_REAL;	(* Position where the search process ends *)
		eEdgeDirection	:	ETcVnEdgeDirection;	(* Specification of the edge direction from aStartPoint to aEndPoint to search for *)
		fMinStrength	:	REAL;	(* Specification of the minimum strength (intensity difference) of the edge to search for *)
		nSearchLines	:	UDINT;	(* Width of the search window, i.e. the number of search lines (1, 3, 5, 7, ...), centered around the line specified by aStartPoint and aEndPoint *)
		fSearchLineDist	:	REAL;	(* Distance between the search lines in pixels (> 0) *)
		nMaxThickness	:	UDINT;	(* Specification of the maximum thickness of the edge to search for, which means fMinStrength must be reached within nMaxThickness pixels *)
		bInvertSearchDirection	:	BOOL;	(* If true, the search starts from the center point between aStartPoint and aEndPoint in both directions *)
		fSearchGap	:	REAL;	(* Optional width of a gap (>= 0, centered between aStartPoint and aEndPoint), that is neglected for searching edges (can reduce execution time). The 2 edges to search for must be on different sides of the gap. *)
		nSubpixelsIterations	:	UDINT;	(* Specifies the number of subpixels (for INTERPOLATION, 10 - 20 usually is sufficient) or maximum number of iterations for optimizing the parameters (for APPROX_ERF and APPROX_GAUSSIAN, 100 usually is sufficient) *)
		fApproxPrecision	:	REAL;	(* Specifies the approximation precision for APPROX_ERF and APPROX_GAUSSIAN (0.0001 usually is sufficient, unused for INTERPOLATION) *)
		eAlgorithm	:	ETcVnEdgeDetectionAlgorithm;	(* Selection of the edge detection algorithm *)
		ipEdgePoints1	:	REFERENCE TO ITcVnContainer;	(* Returns the detected edge points of the edge near aStartPoint (optional, set to 0 if not required; ContainerType_Vector_TcVnPoint2_REAL) *)
		ipEdgePoints2	:	REFERENCE TO ITcVnContainer;	(* Returns the detected edge points of the edge near aEndPoint (optional, set to 0 if not required; ContainerType_Vector_TcVnPoint2_REAL) *)
		ipDistances	:	REFERENCE TO ITcVnContainer;	(* Returns the distances between the detected edge points (optional, set to 0 if not required; ContainerType_Vector_REAL) *)
		hrPrev	:	HRESULT;	(* HRESULT indicating the result of previous operations (If SUCCEEDED(hrPrev) equals false, no operation is executed.) *)
	END_VAR

END_FUNCTION

// Functions/Measurement/F_VN_MeasureMinEdgeDistance

	{attribute 'TcIecLibraryType'}
	{attribute 'external_name' := 'F_VN_MeasureMinEdgeDistance_GUID_C13DF744_C11F_56C3_6112_0877D1909C51'}
	(* Measure the minimum distance within the specified search window between 2 edges, using an interpolation method. *)
	FUNCTION F_VN_MeasureMinEdgeDistance : HRESULT
	VAR_INPUT
		ipSrcImage	:	ITcVnImage;	(* Source image (1 channel) *)
		fMinDistance	:	REFERENCE TO REAL;	(* Returns the minimum distance between the detected edges *)
		aStartPoint	:	REFERENCE TO TcVnPoint2_REAL;	(* Position from which to start the search process (in the direction of aEndPoint) *)
		aEndPoint	:	REFERENCE TO TcVnPoint2_REAL;	(* Position where the search process ends *)
		eEdgeDirection	:	ETcVnEdgeDirection;	(* Specification of the edge direction from aStartPoint to aEndPoint to search for *)
		fMinStrength	:	REAL;	(* Specification of the minimum strength (intensity difference) of the edge to search for *)
		nSearchLines	:	UDINT;	(* Width of the search window, i.e. the number of search lines (1, 3, 5, 7, ...), centered around the line specified by aStartPoint and aEndPoint *)
		hrPrev	:	HRESULT;	(* HRESULT indicating the result of previous operations (If SUCCEEDED(hrPrev) equals false, no operation is executed.) *)
	END_VAR

END_FUNCTION

// Functions/Measurement/F_VN_MeasureMinEdgeDistanceExp

	{attribute 'TcIecLibraryType'}
	{attribute 'external_name' := 'F_VN_MeasureMinEdgeDistanceExp_GUID_7790676D_E3D2_5105_6F0F_BB14EF31FFA6'}
	(* Measure the minimum distance within the specified search window between 2 edges. (expert function) *)
	FUNCTION F_VN_MeasureMinEdgeDistanceExp : HRESULT
	VAR_INPUT
		ipSrcImage	:	ITcVnImage;	(* Source image (1 channel) *)
		fMinDistance	:	REFERENCE TO REAL;	(* Returns the minimum distance between the detected edges *)
		aStartPoint	:	REFERENCE TO TcVnPoint2_REAL;	(* Position from which to start the search process (in the direction of aEndPoint) *)
		aEndPoint	:	REFERENCE TO TcVnPoint2_REAL;	(* Position where the search process ends *)
		eEdgeDirection	:	ETcVnEdgeDirection;	(* Specification of the edge direction from aStartPoint to aEndPoint to search for *)
		fMinStrength	:	REAL;	(* Specification of the minimum strength (intensity difference) of the edge to search for *)
		nSearchLines	:	UDINT;	(* Width of the search window, i.e. the number of search lines (1, 3, 5, 7, ...), centered around the line specified by aStartPoint and aEndPoint *)
		fSearchLineDist	:	REAL;	(* Distance between the search lines in pixels (> 0) *)
		nMaxThickness	:	UDINT;	(* Specification of the maximum thickness of the edge to search for, which means fMinStrength must be reached within nMaxThickness pixels *)
		bInvertSearchDirection	:	BOOL;	(* If true, the search starts from the center point between aStartPoint and aEndPoint in both directions *)
		fSearchGap	:	REAL;	(* Optional width of a gap (>= 0, centered between aStartPoint and aEndPoint), that is neglected for searching edges (can reduce execution time). The 2 edges to search for must be on different sides of the gap. *)
		nSubpixelsIterations	:	UDINT;	(* Specifies the number of subpixels (for INTERPOLATION, 10 - 20 usually is sufficient) or maximum number of iterations for optimizing the parameters (for APPROX_ERF and APPROX_GAUSSIAN, 100 usually is sufficient) *)
		fApproxPrecision	:	REAL;	(* Specifies the approximation precision for APPROX_ERF and APPROX_GAUSSIAN (0.0001 usually is sufficient, unused for INTERPOLATION) *)
		eAlgorithm	:	ETcVnEdgeDetectionAlgorithm;	(* Selection of the edge detection algorithm *)
		ipEdgePoints1	:	REFERENCE TO ITcVnContainer;	(* Returns the detected edge points of the edge near aStartPoint (optional, set to 0 if not required; ContainerType_Vector_TcVnPoint2_REAL) *)
		ipEdgePoints2	:	REFERENCE TO ITcVnContainer;	(* Returns the detected edge points of the edge near aEndPoint (optional, set to 0 if not required; ContainerType_Vector_TcVnPoint2_REAL) *)
		aPoint1	:	REFERENCE TO TcVnPoint2_REAL;	(* Returns the point on the edge near aStartPoint, for which the minimum distance is achieved *)
		aPoint2	:	REFERENCE TO TcVnPoint2_REAL;	(* Returns the point on the edge near aEndPoint, for which the minimum distance is achieved *)
		hrPrev	:	HRESULT;	(* HRESULT indicating the result of previous operations (If SUCCEEDED(hrPrev) equals false, no operation is executed.) *)
	END_VAR

END_FUNCTION

// Functions/Basic Container Operations/F_VN_AdvanceIterator

	{attribute 'TcIecLibraryType'}
	{attribute 'external_name' := 'F_VN_AdvanceIterator_GUID_D71FA0EC_CC29_5059_5665_2D8152FD9A34'}
	(* Advance an iterator by the specified offset. *)
	FUNCTION F_VN_AdvanceIterator : HRESULT
	VAR_INPUT
		ipIterator	:	ITcVnForwardIterator;	(* Iterator to be advanced *)
		nOffset	:	LINT;	(* Offset, by which ipIterator is advanced *)
		hrPrev	:	HRESULT;	(* HRESULT indicating the result of previous operations (If SUCCEEDED(hrPrev) equals false, no operation is executed.) *)
	END_VAR

END_FUNCTION

// Functions/Basic Container Operations/F_VN_CheckIfEmpty

	{attribute 'TcIecLibraryType'}
	{attribute 'external_name' := 'F_VN_CheckIfEmpty_GUID_8CFDD9DC_A17B_5BD0_6341_06CA12108EF6'}
	(* Checks if the container is empty. (Alternatively use interface method .CheckIfEmpty.) *)
	FUNCTION F_VN_CheckIfEmpty : HRESULT
	VAR_INPUT
		ipContainer	:	ITcVnContainer;	(* Container *)
		hrPrev	:	HRESULT;	(* HRESULT indicating the result of previous operations (If SUCCEEDED(hrPrev) equals false, no operation is executed.) *)
	END_VAR

END_FUNCTION

// Functions/Basic Container Operations/F_VN_CheckIfIteratorIsAtEnd

	{attribute 'TcIecLibraryType'}
	{attribute 'external_name' := 'F_VN_CheckIfIteratorIsAtEnd_GUID_4B158961_2402_5B63_78C9_87B9FFF412B5'}
	(* Checks if the iterator points to the past-the-end element. (Alternatively use interface method .CheckIfEnd.) *)
	FUNCTION F_VN_CheckIfIteratorIsAtEnd : HRESULT
	VAR_INPUT
		ipIterator	:	ITcVnForwardIterator;	(* Iterator *)
		hrPrev	:	HRESULT;	(* HRESULT indicating the result of previous operations (If SUCCEEDED(hrPrev) equals false, no operation is executed.) *)
	END_VAR

END_FUNCTION

// Functions/Basic Container Operations/F_VN_ConvertContainerType

	{attribute 'TcIecLibraryType'}
	{attribute 'external_name' := 'F_VN_ConvertContainerType_GUID_7A76B4FB_CCC0_5C89_524E_BABD62E2632E'}
	(* Converts a container to another type (The element type is limited to non-container types, in particular, arithmetic types and arrays). *)
	FUNCTION F_VN_ConvertContainerType : HRESULT
	VAR_INPUT
		ipSrcContainer	:	ITcVnContainer;	(* Source container *)
		ipDestContainer	:	REFERENCE TO ITcVnContainer;	(* Returns the converted container *)
		nDestTypeGuid	:	GUID;	(* Specifies the destination container type for the conversion *)
		hrPrev	:	HRESULT;	(* HRESULT indicating the result of previous operations (If SUCCEEDED(hrPrev) equals false, no operation is executed.) *)
	END_VAR

END_FUNCTION

// Functions/Basic Container Operations/F_VN_CopyContainer

	{attribute 'TcIecLibraryType'}
	{attribute 'external_name' := 'F_VN_CopyContainer_GUID_A174EA54_0A6E_5F4B_4CDA_0A24FB5E7AC5'}
	(* Copys a container. *)
	FUNCTION F_VN_CopyContainer : HRESULT
	VAR_INPUT
		ipSrcContainer	:	ITcVnContainer;	(* Source container *)
		ipDestContainer	:	REFERENCE TO ITcVnContainer;	(* Destination container (same type ID as ipSrcContainer; Non-zero interface pointers are reused.) *)
		hrPrev	:	HRESULT;	(* HRESULT indicating the result of previous operations (If SUCCEEDED(hrPrev) equals false, no operation is executed.) *)
	END_VAR

END_FUNCTION

// Functions/Basic Container Operations/F_VN_CopyContainerElementsConditional_ITcVnContainer

	{attribute 'TcIecLibraryType'}
	{attribute 'external_name' := 'F_VN_CopyContainerElementsConditional_ITcVnContainer_GUID_54910489_26CC_5FAC_7D6E_8ABCBD2E25BB'}
	(* Copys container elements to a new container, depending on a custom condition. *)
	FUNCTION F_VN_CopyContainerElementsConditional_ITcVnContainer : HRESULT
	VAR_INPUT
		ipSrcContainer	:	ITcVnContainer;	(* Source container *)
		ipDestContainer	:	REFERENCE TO ITcVnContainer;	(* Returns a container with elements, that match the condition *)
		ipConditionFB	:	ITcVnCustomElementCondition_ITcVnContainer;	(* Custom condition *)
		hrPrev	:	HRESULT;	(* HRESULT indicating the result of previous operations (If SUCCEEDED(hrPrev) equals false, no operation is executed.) *)
	END_VAR

END_FUNCTION

// Interfaces/Containers/Function Blocks/ITcVnCustomElementCondition_ITcVnContainer

	(* Offers an interface for a custom condition computed for a container. *)
	{attribute 'c++_compatible'}
	INTERFACE ITcVnCustomElementCondition_ITcVnContainer


(* Evaluates the condition for the container. *)
	{attribute 'c++_compatible'}
	{attribute 'minimal_input_size' := '4'}
	{attribute 'pack_mode' := '4'}
	METHOD Condition : BOOL
	VAR_INPUT
		ipElement : ITcVnContainer;
	END_VAR
END_METHOD

END_INTERFACE

// Functions/Basic Container Operations/F_VN_CopyContainerElementsConditional_ITcVnForwardIterator

	{attribute 'TcIecLibraryType'}
	{attribute 'external_name' := 'F_VN_CopyContainerElementsConditional_ITcVnForwardIterator_GUID_388B5F98_F2EC_59C1_7A67_69B6B14C5293'}
	(* Copys container elements to a new container, depending on a custom condition. *)
	FUNCTION F_VN_CopyContainerElementsConditional_ITcVnForwardIterator : HRESULT
	VAR_INPUT
		ipSrcContainer	:	ITcVnContainer;	(* Source container *)
		ipDestContainer	:	REFERENCE TO ITcVnContainer;	(* Returns a container with elements, that match the condition *)
		ipConditionFB	:	ITcVnCustomElementCondition_ITcVnForwardIterator;	(* Custom condition *)
		hrPrev	:	HRESULT;	(* HRESULT indicating the result of previous operations (If SUCCEEDED(hrPrev) equals false, no operation is executed.) *)
	END_VAR

END_FUNCTION

// Interfaces/Containers/Function Blocks/ITcVnCustomElementCondition_ITcVnForwardIterator

	(* Offers an interface for a custom condition computed for an element represented by an ITcVnForwardIterator. *)
	{attribute 'c++_compatible'}
	INTERFACE ITcVnCustomElementCondition_ITcVnForwardIterator


(* Evaluates the condition for the provided element. *)
	{attribute 'c++_compatible'}
	{attribute 'minimal_input_size' := '4'}
	{attribute 'pack_mode' := '4'}
	METHOD Condition : BOOL
	VAR_INPUT
		ipElement : ITcVnForwardIterator;
	END_VAR
END_METHOD

END_INTERFACE

// Functions/Basic Container Operations/F_VN_CreateContainer

	{attribute 'TcIecLibraryType'}
	{attribute 'external_name' := 'F_VN_CreateContainer_GUID_1A043082_9ED9_5B26_60D7_012195767DE6'}
	(* Creates a container with type GUID nTypeGuid and return its container interface. *)
	FUNCTION F_VN_CreateContainer : HRESULT
	VAR_INPUT
		ipContainer	:	REFERENCE TO ITcVnContainer;	(* Returns the created container *)
		nTypeGuid	:	GUID;	(* Type GUID of the container to be created *)
		nElementNum	:	ULINT;	(* Number of elements *)
		hrPrev	:	HRESULT;	(* HRESULT indicating the result of previous operations (If SUCCEEDED(hrPrev) equals false, no operation is executed.) *)
	END_VAR

END_FUNCTION

// Functions/Basic Container Operations/F_VN_CreateContainerFromArray

	{attribute 'TcIecLibraryType'}
	{attribute 'external_name' := 'F_VN_CreateContainerFromArray_GUID_D18C744E_5465_57D7_4907_F87541C57727'}
	(* Creates a container with type GUID nTypeGuid, initialize it with provided data and return its container interface. Only supported for basic container types, i.e. not for containers of containers. *)
	FUNCTION F_VN_CreateContainerFromArray : HRESULT
	VAR_INPUT
		pData	:	PVOID;	(* Pointer to the data array. Make sure that the array contains at least nElementNum elements and that the array element type matches the container element type. *)
		ipContainer	:	REFERENCE TO ITcVnContainer;	(* Returns the created container *)
		nTypeGuid	:	GUID;	(* Type GUID of the container to be created *)
		nElementNum	:	ULINT;	(* Number of elements to copy from pData *)
		hrPrev	:	HRESULT;	(* HRESULT indicating the result of previous operations (If SUCCEEDED(hrPrev) equals false, no operation is executed.) *)
	END_VAR

END_FUNCTION

// Functions/Basic Container Operations/F_VN_EraseFromContainer

	{attribute 'TcIecLibraryType'}
	{attribute 'external_name' := 'F_VN_EraseFromContainer_GUID_AD510B8A_5AA3_5461_6B79_EA807A1724CF'}
	(* Erase elements from a container. *)
	FUNCTION F_VN_EraseFromContainer : HRESULT
	VAR_INPUT
		ipContainer	:	ITcVnContainer;	(* Container from which to erase elements *)
		nStartIdx	:	ULINT;	(* Index of the first element to erase *)
		nCount	:	ULINT;	(* Number of elements to erase *)
		hrPrev	:	HRESULT;	(* HRESULT indicating the result of previous operations (If SUCCEEDED(hrPrev) equals false, no operation is executed.) *)
	END_VAR

END_FUNCTION

// Functions/Basic Container Operations/F_VN_ExportContainer

	{attribute 'TcIecLibraryType'}
	{attribute 'external_name' := 'F_VN_ExportContainer_GUID_C8C71479_CC4E_55A8_5D62_42B38AF34217'}
	(* Export the container elements into a buffer (e.g. an array). Only possible for containers with basic elements. *)
	FUNCTION F_VN_ExportContainer : HRESULT
	VAR_INPUT
		ipContainer	:	ITcVnContainer;	(* Container with basic elements *)
		pBuffer	:	PVOID;	(* Buffer to store the container elements (Make sure to allocate enough memory! The required size in bytes can be determined using the function F_VN_ExportContainerSize) *)
		nBufferSize	:	ULINT;	(* Size of the buffer memory in bytes *)
		hrPrev	:	HRESULT;	(* HRESULT indicating the result of previous operations (If SUCCEEDED(hrPrev) equals false, no operation is executed.) *)
	END_VAR

END_FUNCTION

// Functions/Basic Container Operations/F_VN_ExportContainerSize

	{attribute 'TcIecLibraryType'}
	{attribute 'external_name' := 'F_VN_ExportContainerSize_GUID_0D23F224_EE10_5AEB_5062_811832C44F57'}
	(* Determine the required buffer size in bytes to store all container elements (number_of_Elements * size_per_Element). Only possible for containers with basic elements. *)
	FUNCTION F_VN_ExportContainerSize : HRESULT
	VAR_INPUT
		ipContainer	:	ITcVnContainer;	(* Container with basic elements *)
		nBufferSize	:	REFERENCE TO ULINT;	(* Output parameter containing the required buffer size *)
		hrPrev	:	HRESULT;	(* HRESULT indicating the result of previous operations (If SUCCEEDED(hrPrev) equals false, no operation is executed.) *)
	END_VAR

END_FUNCTION

// Functions/Basic Container Operations/F_VN_ExportContainer_String

	{attribute 'TcIecLibraryType'}
	{attribute 'external_name' := 'F_VN_ExportContainer_String_GUID_200FE250_4F75_5BC2_6922_695CBFB42ABC'}
	(* Export the container elements into a string. Only possible for containers of type ContainerType_String_SINT. *)
	FUNCTION F_VN_ExportContainer_String : HRESULT
	VAR_INPUT
		ipContainer	:	ITcVnContainer;	(* Container of type ContainerType_String_SINT *)
	END_VAR
	VAR_IN_OUT CONSTANT
		sText	:	STRING;	(* Make sure to choose a sufficient STRING size! The required size can be determined using the function VnExportContainerSize. *)
	END_VAR
	VAR_INPUT
		nMaxLength	:	ULINT;	(* Maximum string length to export (including 0 termination). If the container content is longer, the string is cut off at nMaxLength - 1 and 0 termination is appended. In this case, S_FALSE is returned. *)
		hrPrev	:	HRESULT;	(* HRESULT indicating the result of previous operations (If SUCCEEDED(hrPrev) equals false, no operation is executed.) *)
	END_VAR

END_FUNCTION

// Functions/Basic Container Operations/F_VN_ExportSubContainer

	{attribute 'TcIecLibraryType'}
	{attribute 'external_name' := 'F_VN_ExportSubContainer_GUID_57A19812_99CE_574D_7FEF_3BB1DA20A22E'}
	(* Export the container elements of a sub-container into a buffer (e.g. an array). Only possible for 2-dimensional containers with basic elements. *)
	FUNCTION F_VN_ExportSubContainer : HRESULT
	VAR_INPUT
		ipContainer	:	ITcVnContainer;	(* Container with basic elements *)
		nIndex	:	ULINT;	(* Index of the requested element *)
		pBuffer	:	PVOID;	(* Buffer to store the container elements (Make sure to allocate enough memory! The required size in bytes can be determined using the function F_VN_ExportSubContainerSize) *)
		nBufferSize	:	ULINT;	(* Size of the buffer memory in bytes *)
		hrPrev	:	HRESULT;	(* HRESULT indicating the result of previous operations (If SUCCEEDED(hrPrev) equals false, no operation is executed.) *)
	END_VAR

END_FUNCTION

// Functions/Basic Container Operations/F_VN_ExportSubContainerSize

	{attribute 'TcIecLibraryType'}
	{attribute 'external_name' := 'F_VN_ExportSubContainerSize_GUID_E1E0C8E2_6A5B_58ED_4EA9_B4CD79957D9E'}
	(* Determine the required buffer size in bytes to store all container elements of a sub-container (number_of_Elements * size_per_Element). Only possible for 2-dimensional containers with basic elements. *)
	FUNCTION F_VN_ExportSubContainerSize : HRESULT
	VAR_INPUT
		ipContainer	:	ITcVnContainer;	(* Container with basic elements *)
		nIndex	:	ULINT;	(* Index of the requested element *)
		nBufferSize	:	REFERENCE TO ULINT;	(* Output parameter containing the required buffer size *)
		hrPrev	:	HRESULT;	(* HRESULT indicating the result of previous operations (If SUCCEEDED(hrPrev) equals false, no operation is executed.) *)
	END_VAR

END_FUNCTION

// Functions/Basic Container Operations/F_VN_ExportSubContainer_String

	{attribute 'TcIecLibraryType'}
	{attribute 'external_name' := 'F_VN_ExportSubContainer_String_GUID_34821399_A303_55DE_4DFF_35BFF6BA6B01'}
	(* Export the container elements of a sub-container into a string. Only possible for 2-dimensional containers of type ContainerType_Vector_String_SINT. *)
	FUNCTION F_VN_ExportSubContainer_String : HRESULT
	VAR_INPUT
		ipContainer	:	ITcVnContainer;	(* Container of type ContainerType_Vector_String_SINT *)
		nIndex	:	ULINT;	(* Index of the requested element *)
	END_VAR
	VAR_IN_OUT CONSTANT
		sText	:	STRING;	(* Make sure to choose a sufficient STRING size! The required size can be determined using the function VnExportSubContainerSize. *)
	END_VAR
	VAR_INPUT
		nMaxLength	:	ULINT;	(* Maximum string length to export (including 0 termination). If the container content is longer, the string is cut off at nMaxLength - 1 and 0 termination is appended. In this case, S_FALSE is returned. *)
		hrPrev	:	HRESULT;	(* HRESULT indicating the result of previous operations (If SUCCEEDED(hrPrev) equals false, no operation is executed.) *)
	END_VAR

END_FUNCTION

// Functions/Basic Container Operations/F_VN_ExtractContainerRange

	{attribute 'TcIecLibraryType'}
	{attribute 'external_name' := 'F_VN_ExtractContainerRange_GUID_3565CD79_5F87_5175_6E1D_46C90C1E8C86'}
	(* Copy the specified range of the source container into the destination container. (If the destination container already contains elements, they will be removed.) *)
	FUNCTION F_VN_ExtractContainerRange : HRESULT
	VAR_INPUT
		ipSrcContainer	:	ITcVnContainer;	(* Source container *)
		ipDestContainer	:	REFERENCE TO ITcVnContainer;	(* Destination container *)
		nFirstIdx	:	ULINT;	(* Index of the first element to copy *)
		nLastIdx	:	ULINT;	(* Index of the last element to copy *)
		hrPrev	:	HRESULT;	(* HRESULT indicating the result of previous operations (If SUCCEEDED(hrPrev) equals false, no operation is executed.) *)
	END_VAR

END_FUNCTION

// Functions/Basic Container Operations/F_VN_GetContainer

	{attribute 'TcIecLibraryType'}
	{attribute 'external_name' := 'F_VN_GetContainer_GUID_5C8712FF_CA7A_549B_6819_A3ED3B1CA12D'}
	(* Gets a pointer to the current element converted into an ITcVnContainer interface and increment its reference counter (only possible for container types). (Alternatively use interface method .GetContainer.) *)
	FUNCTION F_VN_GetContainer : HRESULT
	VAR_INPUT
		ipIterator	:	ITcVnForwardIterator;	(* Iterator *)
		ipContainer	:	REFERENCE TO ITcVnContainer;	(* Returns the container interface *)
		hrPrev	:	HRESULT;	(* HRESULT indicating the result of previous operations (If SUCCEEDED(hrPrev) equals false, no operation is executed.) *)
	END_VAR

END_FUNCTION

// Functions/Basic Container Operations/F_VN_GetContainerExp

	{attribute 'TcIecLibraryType'}
	{attribute 'external_name' := 'F_VN_GetContainerExp_GUID_38BBB872_A787_5425_42D9_A82091BBD1CD'}
	(* Gets a pointer to the current element converted into an ITcVnContainer interface and increment its reference counter (only possible for container types). Additionally, an offset to increment or decrement the iterator afterwards can be provided. (expert function) *)
	FUNCTION F_VN_GetContainerExp : HRESULT
	VAR_INPUT
		ipIterator	:	ITcVnForwardIterator;	(* Iterator *)
		ipContainer	:	REFERENCE TO ITcVnContainer;	(* Returns the container interface *)
		nOffset	:	DINT;	(* Offset to increment (>0) or decrement (<0) the iterator afterwards *)
		hrPrev	:	HRESULT;	(* HRESULT indicating the result of previous operations (If SUCCEEDED(hrPrev) equals false, no operation is executed.) *)
	END_VAR

END_FUNCTION

// Functions/Basic Container Operations/F_VN_GetForwardIterator

	{attribute 'TcIecLibraryType'}
	{attribute 'external_name' := 'F_VN_GetForwardIterator_GUID_38D0C6E1_0365_5285_7B85_9BAECF49C284'}
	(* Gets a forward iterator for the container. (Alternatively use interface method .GetForwardIterator.) *)
	FUNCTION F_VN_GetForwardIterator : HRESULT
	VAR_INPUT
		ipContainer	:	ITcVnContainer;	(* Container *)
		ipIterator	:	REFERENCE TO ITcVnForwardIterator;	(* Returns the iterator interface *)
		hrPrev	:	HRESULT;	(* HRESULT indicating the result of previous operations (If SUCCEEDED(hrPrev) equals false, no operation is executed.) *)
	END_VAR

END_FUNCTION

// Functions/Basic Container Operations/F_VN_GetNumberOfElements

	{attribute 'TcIecLibraryType'}
	{attribute 'external_name' := 'F_VN_GetNumberOfElements_GUID_BABF0399_9F8D_5539_4882_19251BACFFCF'}
	(* Gets the number of elements in the container. (Alternatively use interface method .getElementNum.) *)
	FUNCTION F_VN_GetNumberOfElements : HRESULT
	VAR_INPUT
		ipContainer	:	ITcVnContainer;	(* Container *)
		nNumberOfElements	:	REFERENCE TO ULINT;	(* Returns the number of elements in ipContainer *)
		hrPrev	:	HRESULT;	(* HRESULT indicating the result of previous operations (If SUCCEEDED(hrPrev) equals false, no operation is executed.) *)
	END_VAR

END_FUNCTION

// Functions/Basic Container Operations/F_VN_GetRandomAccessIterator

	{attribute 'TcIecLibraryType'}
	{attribute 'external_name' := 'F_VN_GetRandomAccessIterator_GUID_447E6AD1_333C_5FDC_4D03_05157CFA0A81'}
	(* Gets a random access iterator for the container. (Alternatively use interface method .GetRandomAccessIterator.) *)
	FUNCTION F_VN_GetRandomAccessIterator : HRESULT
	VAR_INPUT
		ipContainer	:	ITcVnContainer;	(* Container *)
		ipIterator	:	REFERENCE TO ITcVnRandomAccessIterator;	(* Returns the iterator interface *)
		hrPrev	:	HRESULT;	(* HRESULT indicating the result of previous operations (If SUCCEEDED(hrPrev) equals false, no operation is executed.) *)
	END_VAR

END_FUNCTION

// Functions/Basic Container Operations/F_VN_IncrementIterator

	{attribute 'TcIecLibraryType'}
	{attribute 'external_name' := 'F_VN_IncrementIterator_GUID_12762337_0B81_5978_5D04_BAEEF4371982'}
	(* Increment the iterator. (Alternatively use interface method .Increment.) *)
	FUNCTION F_VN_IncrementIterator : HRESULT
	VAR_INPUT
		ipIterator	:	ITcVnForwardIterator;	(* Iterator *)
		hrPrev	:	HRESULT;	(* HRESULT indicating the result of previous operations (If SUCCEEDED(hrPrev) equals false, no operation is executed.) *)
	END_VAR

END_FUNCTION

// Functions/Basic Container Operations/F_VN_IteratorDistance

	{attribute 'TcIecLibraryType'}
	{attribute 'external_name' := 'F_VN_IteratorDistance_GUID_A7C770BA_2DB1_5B23_620D_FE138273D014'}
	(* Computes the distance between 2 iterators. *)
	FUNCTION F_VN_IteratorDistance : HRESULT
	VAR_INPUT
		ipIteratorFirst	:	ITcVnForwardIterator;	(* First iterator *)
		ipIteratorLast	:	ITcVnForwardIterator;	(* Last iterator *)
		nDistance	:	REFERENCE TO LINT;	(* Returns the computed distance *)
		hrPrev	:	HRESULT;	(* HRESULT indicating the result of previous operations (If SUCCEEDED(hrPrev) equals false, no operation is executed.) *)
	END_VAR

END_FUNCTION

// Functions/Basic Container Operations/F_VN_ReserveContainerMemory

	{attribute 'TcIecLibraryType'}
	{attribute 'external_name' := 'F_VN_ReserveContainerMemory_GUID_DD1E2B87_0E45_5AE7_50E0_4CC79AD471BA'}
	(* Reserve container memory (call with maximum required number of elements before manually appending elements for better performance) *)
	FUNCTION F_VN_ReserveContainerMemory : HRESULT
	VAR_INPUT
		ipContainer	:	ITcVnContainer;	(* Container for which to reserve the memory *)
		nElements	:	ULINT;	(* Number of elements for which the container should reserve memory *)
		hrPrev	:	HRESULT;	(* HRESULT indicating the result of previous operations (If SUCCEEDED(hrPrev) equals false, no operation is executed.) *)
	END_VAR

END_FUNCTION

// Functions/Basic Container Operations/F_VN_ReverseContainer

	{attribute 'TcIecLibraryType'}
	{attribute 'external_name' := 'F_VN_ReverseContainer_GUID_4E265B74_6CA9_5773_66A9_C1DA8A148734'}
	(* Reverse the container elements. *)
	FUNCTION F_VN_ReverseContainer : HRESULT
	VAR_INPUT
		ipContainer	:	ITcVnContainer;	(* Container to be reversed *)
		hrPrev	:	HRESULT;	(* HRESULT indicating the result of previous operations (If SUCCEEDED(hrPrev) equals false, no operation is executed.) *)
	END_VAR

END_FUNCTION

// Functions/Basic Container Operations/F_VN_SetContainer

	{attribute 'TcIecLibraryType'}
	{attribute 'external_name' := 'F_VN_SetContainer_GUID_984433B4_8158_555D_4492_F570F5CD5834'}
	(* Sets the current element using an ITcVnContainer interface (only possible for container types). (Alternatively use interface method .SetContainer.) *)
	FUNCTION F_VN_SetContainer : HRESULT
	VAR_INPUT
		ipIterator	:	ITcVnForwardIterator;	(* Iterator *)
		ipContainer	:	ITcVnContainer;	(* Container interface of which the content is to be assigned to the current element *)
		hrPrev	:	HRESULT;	(* HRESULT indicating the result of previous operations (If SUCCEEDED(hrPrev) equals false, no operation is executed.) *)
	END_VAR

END_FUNCTION

// Functions/Basic Container Operations/F_VN_SetIteratorToBegin

	{attribute 'TcIecLibraryType'}
	{attribute 'external_name' := 'F_VN_SetIteratorToBegin_GUID_2A339118_BAC3_5935_7710_152E4E8346DC'}
	(* Sets the iterator to the first element of the container. (Alternatively use interface method .SetToBegin.) *)
	FUNCTION F_VN_SetIteratorToBegin : HRESULT
	VAR_INPUT
		ipIterator	:	ITcVnForwardIterator;	(* Iterator *)
		hrPrev	:	HRESULT;	(* HRESULT indicating the result of previous operations (If SUCCEEDED(hrPrev) equals false, no operation is executed.) *)
	END_VAR

END_FUNCTION

// Functions/Image Color and Contrast Processing/F_VN_ApplyColorMap

	{attribute 'TcIecLibraryType'}
	{attribute 'external_name' := 'F_VN_ApplyColorMap_GUID_E9586DFF_09FC_52DF_6C1F_FB8E2B6F9D6D'}
	(* Apply a color map to a gray-level image. *)
	FUNCTION F_VN_ApplyColorMap : HRESULT
	VAR_INPUT
		ipSrcImage	:	ITcVnImage;	(* Source image (TCVN_ET_USINT or TCVN_ET_UINT, 1 channel) *)
		ipDestImage	:	REFERENCE TO ITcVnImage;	(* Returns the colored image (TCVN_ET_USINT, 3 channel. An appropriate image will be created if required.) *)
		ipColorMap	:	ITcVnContainer;	(* Color map to be applied to ipSrcImage (ContainerType_Vector_TcVnVector3_REAL with 256 or 65536 elements, dependent on ipSrcImage type). Can be either custom or created with F_VN_GenerateColorMap. *)
		hrPrev	:	HRESULT;	(* HRESULT indicating the result of previous operations (If SUCCEEDED(hrPrev) equals false, no operation is executed.) *)
	END_VAR

END_FUNCTION

// Functions/Image Color and Contrast Processing/F_VN_GenerateColorMap

	{attribute 'TcIecLibraryType'}
	{attribute 'external_name' := 'F_VN_GenerateColorMap_GUID_F78BD2BF_303C_5BB0_474C_8B18359F87EA'}
	(* Generates a pre-defined color map. *)
	FUNCTION F_VN_GenerateColorMap : HRESULT
	VAR_INPUT
		ipColorMap	:	REFERENCE TO ITcVnContainer;	(* Returns the color map (ContainerType_Vector_TcVnVector3_REAL with 256 or 65536 elements) *)
		eColorMap	:	ETcVnColorMap;	(* Selects a color map (similar to GNU Octave/MATLAB types) *)
		eColorMapSize	:	ETcVnColorMapSize;	(* Defines how many elements the generated color map should have *)
		hrPrev	:	HRESULT;	(* HRESULT indicating the result of previous operations (If SUCCEEDED(hrPrev) equals false, no operation is executed.) *)
	END_VAR

END_FUNCTION

// Functions/Image Color and Contrast Processing/F_VN_ConvertColorSpace

	{attribute 'TcIecLibraryType'}
	{attribute 'external_name' := 'F_VN_ConvertColorSpace_GUID_8FB1759A_0046_562B_604A_3EAA995C0B69'}
	(* Convert image from one color space to another. *)
	FUNCTION F_VN_ConvertColorSpace : HRESULT
	VAR_INPUT
		ipSrcImage	:	ITcVnImage;	(* Source image *)
		ipDestImage	:	REFERENCE TO ITcVnImage;	(* Destination image (An appropriate destination image will be created if required.) *)
		eTransform	:	ETcVnColorSpaceTransform;	(* Transforms to be applied *)
		hrPrev	:	HRESULT;	(* HRESULT indicating the result of previous operations (If SUCCEEDED(hrPrev) equals false, no operation is executed.) *)
	END_VAR

END_FUNCTION

// Functions/Image Color and Contrast Processing/F_VN_GenerateCustomColorMap

	{attribute 'TcIecLibraryType'}
	{attribute 'external_name' := 'F_VN_GenerateCustomColorMap_GUID_93BFCC11_8B51_5B9A_56D0_42A594C4A2ED'}
	(* Generate a custom color map by interpolating between user defined colors (equally distributed, linear for each channel). *)
	FUNCTION F_VN_GenerateCustomColorMap : HRESULT
	VAR_INPUT
		ipColorMap	:	REFERENCE TO ITcVnContainer;	(* Returns the color map (ContainerType_Vector_TcVnVector3_REAL with 256 or 65536 elements) *)
		ipInitialColors	:	ITcVnContainer;	(* User defined colors (ContainerType_Vector_TcVnVector3_REAL, at least 2 elements) *)
		eColorMapSize	:	ETcVnColorMapSize;	(* Defines how many elements the generated color map should have *)
		hrPrev	:	HRESULT;	(* HRESULT indicating the result of previous operations (If SUCCEEDED(hrPrev) equals false, no operation is executed.) *)
	END_VAR

END_FUNCTION

// Functions/Image Color and Contrast Processing/F_VN_Histogram

	{attribute 'TcIecLibraryType'}
	{attribute 'external_name' := 'F_VN_Histogram_GUID_FFFE33FD_2E80_5B54_7678_52E4A583E44D'}
	(* Calculate the (multi-channel) histogram of an image. *)
	FUNCTION F_VN_Histogram : HRESULT
	VAR_INPUT
		ipSrcImage	:	ITcVnImage;	(* Source image *)
		ipDestHistogram	:	REFERENCE TO ITcVnContainer;	(* Returns a container with a multi-channel histogram, where every channel is represented as a vector of UDINT (ContainerType_Vector_Vector_UDINT. Non-zero interface pointers are reused.) *)
		hrPrev	:	HRESULT;	(* HRESULT indicating the result of previous operations (If SUCCEEDED(hrPrev) equals false, no operation is executed.) *)
	END_VAR

END_FUNCTION

// Functions/Image Color and Contrast Processing/F_VN_HistogramExp

	{attribute 'TcIecLibraryType'}
	{attribute 'external_name' := 'F_VN_HistogramExp_GUID_74D45244_C0EF_5C23_50AF_3FC1B5267E15'}
	(* Calculate the (multi-channel) histogram of an image. (expert function) *)
	FUNCTION F_VN_HistogramExp : HRESULT
	VAR_INPUT
		ipSrcImage	:	ITcVnImage;	(* Source image *)
		ipDestHistogram	:	REFERENCE TO ITcVnContainer;	(* Returns a container with a multi-channel histogram, where every channel is represented as a vector of UDINT (ContainerType_Vector_Vector_UDINT. Non-zero interface pointers are reused.) *)
		nBins	:	REFERENCE TO UDINT;	(* Desired number of bins or 0 to keep the default for the corresponding image format (in) and default number of bins (out) *)
		fLowerBound	:	REFERENCE TO LREAL;	(* Lower (inclusive) boundary of the 0-th histogram bin (in), or receive the default if fLowerBound AND fUpperBound are set to 0 (out) *)
		fUpperBound	:	REFERENCE TO LREAL;	(* Upper (exclusive) boundary of the last histogram bin nBins-1 (in), or receive the default if fLowerBound AND fUpperBound are set to 0 (out) *)
		ipMask	:	ITcVnImage;	(* Source image mask (TCVN_ET_USINT, 1 channel. Mask is optional, set to 0 if not required.) *)
		hrPrev	:	HRESULT;	(* HRESULT indicating the result of previous operations (If SUCCEEDED(hrPrev) equals false, no operation is executed.) *)
	END_VAR

END_FUNCTION

// Functions/Image Color and Contrast Processing/F_VN_HistogramEqualization

	{attribute 'TcIecLibraryType'}
	{attribute 'external_name' := 'F_VN_HistogramEqualization_GUID_523E818E_8C72_5EFE_6D14_B2758159A578'}
	(* Equalize the histogram of a grayscale or rgb image, which normalizes the brightness and improves the contrast. *)
	FUNCTION F_VN_HistogramEqualization : HRESULT
	VAR_INPUT
		ipSrcImage	:	ITcVnImage;	(* Source image *)
		ipDestImage	:	REFERENCE TO ITcVnImage;	(* Destination image (An appropriate destination image will be created if required.) *)
		hrPrev	:	HRESULT;	(* HRESULT indicating the result of previous operations (If SUCCEEDED(hrPrev) equals false, no operation is executed.) *)
	END_VAR

END_FUNCTION

// Functions/Image Color and Contrast Processing/F_VN_HistogramEqualizationExp

	{attribute 'TcIecLibraryType'}
	{attribute 'external_name' := 'F_VN_HistogramEqualizationExp_GUID_382D58C4_76B9_51F6_407F_CD93E62F684E'}
	(* Equalize the histogram of a grayscale or color image, which normalizes the brightness and improves the contrast. (expert function) 
	The channel index that should be equalized has to be specified (-1 expects a RGB image, converts it to YCbCr, equalizes the Y channel and converts the image back to RGB).  *)
	FUNCTION F_VN_HistogramEqualizationExp : HRESULT
	VAR_INPUT
		ipSrcImage	:	ITcVnImage;	(* Source image *)
		ipDestImage	:	REFERENCE TO ITcVnImage;	(* Destination image (An appropriate destination image will be created if required.) *)
		nChannelIdx	:	INT;	(* Index of the image channel that should be equalized (-1 expects a RGB image, converts it to YCbCr, equalizes the Y channel and converts the image back to RGB) *)
		hrPrev	:	HRESULT;	(* HRESULT indicating the result of previous operations (If SUCCEEDED(hrPrev) equals false, no operation is executed.) *)
	END_VAR

END_FUNCTION

// Functions/Image Color and Contrast Processing/F_VN_InvertImageColor

	{attribute 'TcIecLibraryType'}
	{attribute 'external_name' := 'F_VN_InvertImageColor_GUID_8125ADF6_1302_513A_635E_B3AA6B0DB765'}
	(* Invert the color of an image.
          For signed integer or negative floating point values, only the signs will be switched.
          If the image contains only positive floating point values, each pixel value is subtracted from the maximum available pixel value (or 1.0, whatever is higher). *)
	FUNCTION F_VN_InvertImageColor : HRESULT
	VAR_INPUT
		ipSrcImage	:	ITcVnImage;	(* Source image *)
		ipDestImage	:	REFERENCE TO ITcVnImage;	(* Destination image (An appropriate image will be created if required.) *)
		hrPrev	:	HRESULT;	(* HRESULT indicating the result of previous operations (If SUCCEEDED(hrPrev) equals false, no operation is executed.) *)
	END_VAR

END_FUNCTION

// Functions/Image Color and Contrast Processing/F_VN_InvertImageColorExp

	{attribute 'TcIecLibraryType'}
	{attribute 'external_name' := 'F_VN_InvertImageColorExp_GUID_6E53BEEC_723A_5190_5011_EF45CE8976A9'}
	(* Invert the color of an image. (expert function)
          For signed integer or negative floating point values, only the signs will be switched.
          If the image contains only positive floating point values, each pixel value is subtracted from the maximum available pixel value (or 1.0, whatever is higher). *)
	FUNCTION F_VN_InvertImageColorExp : HRESULT
	VAR_INPUT
		ipSrcImage	:	ITcVnImage;	(* Source image *)
		ipDestImage	:	REFERENCE TO ITcVnImage;	(* Destination image (An appropriate image will be created if required.) *)
		fMaxValue	:	LREAL;	(* Maximum pixel value (e.g. if a 16 bit image contains 12 bit values). -1 means the default values are used. *)
		hrPrev	:	HRESULT;	(* HRESULT indicating the result of previous operations (If SUCCEEDED(hrPrev) equals false, no operation is executed.) *)
	END_VAR

END_FUNCTION

// Functions/Image Color and Contrast Processing/F_VN_NormalizeImage

	{attribute 'TcIecLibraryType'}
	{attribute 'external_name' := 'F_VN_NormalizeImage_GUID_B750D483_F2AA_5090_5915_8D767E08BEFD'}
	(* Normalize an image regarding its value range (e.g. stretch pixel values [50..150] to full range [0..255]). *)
	FUNCTION F_VN_NormalizeImage : HRESULT
	VAR_INPUT
		ipSrcImage	:	ITcVnImage;	(* Source image *)
		ipDestImage	:	REFERENCE TO ITcVnImage;	(* Destination image (An appropriate destination image will be created if required.) *)
		hrPrev	:	HRESULT;	(* HRESULT indicating the result of previous operations (If SUCCEEDED(hrPrev) equals false, no operation is executed.) *)
	END_VAR

END_FUNCTION

// Functions/Image Color and Contrast Processing/F_VN_NormalizeImageExp

	{attribute 'TcIecLibraryType'}
	{attribute 'external_name' := 'F_VN_NormalizeImageExp_GUID_4FBC936F_B7E6_551A_7C04_2B7B1A3364B1'}
	(* Normalize an image regarding its value range (e.g. stretch pixel values [50..150] to full range [0..255]) or scale the values regarding a specific normalization (e.g. L2-norm). (expert function) *)
	FUNCTION F_VN_NormalizeImageExp : HRESULT
	VAR_INPUT
		ipSrcImage	:	ITcVnImage;	(* Source image *)
		ipDestImage	:	REFERENCE TO ITcVnImage;	(* Destination image (An appropriate destination image will be created if required.) *)
		fAlpha	:	LREAL;	(* Lower range boundary (in case of normalizing the value range) or value to normalize to (||ipDestImage|| = fAlpha) *)
		fBeta	:	LREAL;	(* Upper range boundary (in case of normalizing the value range) *)
		eNormType	:	ETcVnNormalizationType;	(* Normalization type (only INF, L1, L2 or MINMAX) *)
		eDestType	:	ETcVnElementType;	(* Destination image depth (usually SAME_AS_SOURCE) *)
		ipMask	:	ITcVnImage;	(* Mask to restrict the normalization to specific pixel positions (set 0 to normalize the whole image) *)
		hrPrev	:	HRESULT;	(* HRESULT indicating the result of previous operations (If SUCCEEDED(hrPrev) equals false, no operation is executed.) *)
	END_VAR

END_FUNCTION

// Functions/Image Color and Contrast Processing/F_VN_NormalizeImageForDisplay

	{attribute 'TcIecLibraryType'}
	{attribute 'external_name' := 'F_VN_NormalizeImageForDisplay_GUID_ECA03700_3D68_5CCD_5EA6_E50897B64D63'}
	(* Normalize an image for display, i.e. scale it to the full value range of the underlying data type (-1 to 1 for floating point). *)
	FUNCTION F_VN_NormalizeImageForDisplay : HRESULT
	VAR_INPUT
		ipSrcImage	:	ITcVnImage;	(* Source image *)
		ipDestImage	:	REFERENCE TO ITcVnImage;	(* Destination image (An appropriate destination image will be created if required.) *)
		eSignedNormalization	:	ETcVnSignedNormalization;	(* Option for normalizing signed values *)
		hrPrev	:	HRESULT;	(* HRESULT indicating the result of previous operations (If SUCCEEDED(hrPrev) equals false, no operation is executed.) *)
	END_VAR

END_FUNCTION

// Functions/Image Color and Contrast Processing/F_VN_ReferenceColorSimilarity_ITcVnColorModel

	{attribute 'TcIecLibraryType'}
	{attribute 'external_name' := 'F_VN_ReferenceColorSimilarity_ITcVnColorModel_GUID_9C86E25B_95C0_558A_6670_DBD9D206B9EE'}
	(* Computes the similarity to a reference color model for each pixel in the source image. *)
	FUNCTION F_VN_ReferenceColorSimilarity_ITcVnColorModel : HRESULT
	VAR_INPUT
		ipSrcImage	:	ITcVnImage;	(* RGB source image (USINT, 3 channels) *)
		ipDestImage	:	REFERENCE TO ITcVnImage;	(* Returns the similarity to ipColorModel for each pixel in ipSrcImage (USINT, 1 channel. An appropriate destination image will be created if required.) *)
		ipColorModel	:	ITcVnColorModel;	(* Color model *)
		hrPrev	:	HRESULT;	(* HRESULT indicating the result of previous operations (If SUCCEEDED(hrPrev) equals false, no operation is executed.) *)
	END_VAR

END_FUNCTION

// Interfaces/Machine Learning/ITcVnColorModel

	(* Interface to train and classify an image color. *)
	{attribute 'c++_compatible'}
	{attribute 'vtable_order' := 'TrainImageColor;ClassifyImageColor'}
	INTERFACE ITcVnColorModel EXTENDS ITcVnMlModel


(* Train the color of the provided image. *)
	{attribute 'c++_compatible'}
	{attribute 'minimal_input_size' := '4'}
	{attribute 'pack_mode' := '4'}
	METHOD TrainImageColor : HRESULT
	VAR_INPUT
		ipSrcImage : ITcVnImage;
		nDifferentColors : UDINT;
		ipMask : ITcVnImage;
		nSkipPixels : UDINT;
	END_VAR
END_METHOD


(* Compute the similarity of each image pixel to the trained reference color. *)
	{attribute 'c++_compatible'}
	{attribute 'minimal_input_size' := '4'}
	{attribute 'pack_mode' := '4'}
	METHOD ClassifyImageColor : HRESULT
	VAR_INPUT
		ipSrcImage : ITcVnImage;
		pipDestImage : POINTER TO ITcVnImage;
		fVariance : REAL;
		fLuminanceWeight : REAL;
	END_VAR
END_METHOD

END_INTERFACE

// Functions/Image Color and Contrast Processing/F_VN_ReferenceColorSimilarityExp_ITcVnColorModel

	{attribute 'TcIecLibraryType'}
	{attribute 'external_name' := 'F_VN_ReferenceColorSimilarityExp_ITcVnColorModel_GUID_989AD2E0_1C31_543D_4CC9_057C6F1CF89A'}
	(* Computes the similarity to a reference color model for each pixel in the source image. (expert function) *)
	FUNCTION F_VN_ReferenceColorSimilarityExp_ITcVnColorModel : HRESULT
	VAR_INPUT
		ipSrcImage	:	ITcVnImage;	(* RGB source image (USINT, 3 channels) *)
		ipDestImage	:	REFERENCE TO ITcVnImage;	(* Returns the similarity to ipColorModel for each pixel in ipSrcImage (USINT, 1 channel. An appropriate destination image will be created if required.) *)
		ipColorModel	:	ITcVnColorModel;	(* Color model *)
		fVariance	:	REAL;	(* Allowed color variance (0.1 - 0.3 might be a good start to try) *)
		fLuminanceWeight	:	REAL;	(* Weight the impact of the luminance ([0..1], e.g. set to 0 to be more resistant to unequal illumination, but might be required to differentiate between some colors. Ignored if ipColorModel is of type RGB.) *)
		hrPrev	:	HRESULT;	(* HRESULT indicating the result of previous operations (If SUCCEEDED(hrPrev) equals false, no operation is executed.) *)
	END_VAR

END_FUNCTION

// Functions/Image Color and Contrast Processing/F_VN_ReferenceColorSimilarity_TcVnVector3_LREAL

	{attribute 'TcIecLibraryType'}
	{attribute 'external_name' := 'F_VN_ReferenceColorSimilarity_TcVnVector3_LREAL_GUID_4C661328_A4CC_5C7E_59B5_2FCF1B9E2CC1'}
	(* Computes the similarity to a reference color for each pixel in the source image. *)
	FUNCTION F_VN_ReferenceColorSimilarity_TcVnVector3_LREAL : HRESULT
	VAR_INPUT
		ipSrcImage	:	ITcVnImage;	(* RGB source image (USINT, 3 channels) *)
		ipDestImage	:	REFERENCE TO ITcVnImage;	(* Returns the similarity to aRefColor for each pixel in ipSrcImage (USINT, 1 channel. An appropriate destination image will be created if required.) *)
		aRefColor	:	REFERENCE TO TcVnVector3_LREAL;	(* Reference color (RGB, [0..255]) *)
		hrPrev	:	HRESULT;	(* HRESULT indicating the result of previous operations (If SUCCEEDED(hrPrev) equals false, no operation is executed.) *)
	END_VAR

END_FUNCTION

// Functions/Image Color and Contrast Processing/F_VN_ReferenceColorSimilarityExp_TcVnVector3_LREAL

	{attribute 'TcIecLibraryType'}
	{attribute 'external_name' := 'F_VN_ReferenceColorSimilarityExp_TcVnVector3_LREAL_GUID_65ED382D_872A_56AB_6D6D_7CDCF2FFB4D5'}
	(* Computes the similarity to a reference color for each pixel in the source image. (expert function) *)
	FUNCTION F_VN_ReferenceColorSimilarityExp_TcVnVector3_LREAL : HRESULT
	VAR_INPUT
		ipSrcImage	:	ITcVnImage;	(* RGB source image (USINT, 3 channels) *)
		ipDestImage	:	REFERENCE TO ITcVnImage;	(* Returns the similarity to aRefColor for each pixel in ipSrcImage (USINT, 1 channel. An appropriate destination image will be created if required.) *)
		aRefColor	:	REFERENCE TO TcVnVector3_LREAL;	(* Reference color (RGB, [0..255]) *)
		fVariance	:	REAL;	(* Allowed color variance (0.1 - 0.3 might be a good start to try) *)
		fLuminanceWeight	:	REAL;	(* Weight the impact of the luminance ([0..1], e.g. set to 0 to be more resistant to unequal illumination, but might be required to differentiate between some colors) *)
		hrPrev	:	HRESULT;	(* HRESULT indicating the result of previous operations (If SUCCEEDED(hrPrev) equals false, no operation is executed.) *)
	END_VAR

END_FUNCTION

// Functions/Image Color and Contrast Processing/F_VN_TrainImageColor

	{attribute 'TcIecLibraryType'}
	{attribute 'external_name' := 'F_VN_TrainImageColor_GUID_B41F4EC3_A2CC_5CE3_6DE3_F42F70285271'}
	(* Create a new color model, describing the image color. *)
	FUNCTION F_VN_TrainImageColor : HRESULT
	VAR_INPUT
		ipSrcImage	:	ITcVnImage;	(* Source image (3 channels (RGB) of type USINT) *)
		ipColorModel	:	REFERENCE TO ITcVnColorModel;	(* Returns the color model *)
		nDifferentColors	:	UDINT;	(* Number of different colors to distinguish *)
		hrPrev	:	HRESULT;	(* HRESULT indicating the result of previous operations (If SUCCEEDED(hrPrev) equals false, no operation is executed.) *)
	END_VAR

END_FUNCTION

// Functions/Image Color and Contrast Processing/F_VN_TrainImageColorExp

	{attribute 'TcIecLibraryType'}
	{attribute 'external_name' := 'F_VN_TrainImageColorExp_GUID_D7CACD6A_396F_5B91_4AFD_A869A98D7B88'}
	(* Create a new color model, describing the image color. (expert function) *)
	FUNCTION F_VN_TrainImageColorExp : HRESULT
	VAR_INPUT
		ipSrcImage	:	ITcVnImage;	(* Source image (3 channels (RGB) of type USINT) *)
		ipColorModel	:	REFERENCE TO ITcVnColorModel;	(* Returns the color model *)
		nDifferentColors	:	UDINT;	(* Number of different colors to distinguish *)
		eMethod	:	ETcVnColorTrainingMethod;	(* Color training method *)
		ipMask	:	ITcVnImage;	(* Optional image mask (1 channel of type USINT, set to 0 if not required) *)
		nSkipPixels	:	UDINT;	(* Number of pixels to skip between each evaluated color sample (to achieve a better performance). 0 takes every pixel into account and tends to be more accurate. *)
		hrPrev	:	HRESULT;	(* HRESULT indicating the result of previous operations (If SUCCEEDED(hrPrev) equals false, no operation is executed.) *)
	END_VAR

END_FUNCTION

// Functions/Geometric and Coordinate Transformations/F_VN_ApplyRotationToAffineTransformation

	{attribute 'TcIecLibraryType'}
	{attribute 'external_name' := 'F_VN_ApplyRotationToAffineTransformation_GUID_A97DA3CD_9107_51B0_5459_32B6494C0415'}
	(* Apply a rotation to an existing 2D affine transformation matrix. *)
	FUNCTION F_VN_ApplyRotationToAffineTransformation : HRESULT
	VAR_INPUT
		aTransformationMatrix	:	REFERENCE TO TcVnMatrix2x3_LREAL;	(* Affine transformation matrix to which the rotation is applied *)
		fAngle	:	LREAL;	(* Angle in radians (positive means counter-clockwise) *)
		hrPrev	:	HRESULT;	(* HRESULT indicating the result of previous operations (If SUCCEEDED(hrPrev) equals false, no operation is executed.) *)
	END_VAR

END_FUNCTION

// Functions/Geometric and Coordinate Transformations/F_VN_ApplyRotationToAffineTransformationExp

	{attribute 'TcIecLibraryType'}
	{attribute 'external_name' := 'F_VN_ApplyRotationToAffineTransformationExp_GUID_72565882_D705_5353_47D9_C1B5DFEC9E4D'}
	(* Apply a rotation to an existing 2D affine transformation matrix. (expert function) *)
	FUNCTION F_VN_ApplyRotationToAffineTransformationExp : HRESULT
	VAR_INPUT
		aTransformationMatrix	:	REFERENCE TO TcVnMatrix2x3_LREAL;	(* Affine transformation matrix to which the rotation is applied *)
		fAngle	:	LREAL;	(* Angle in radians (positive means counter-clockwise) *)
		bUsePreMultiplication	:	BOOL;	(* Select if pre- or post-multiplication should be used *)
		hrPrev	:	HRESULT;	(* HRESULT indicating the result of previous operations (If SUCCEEDED(hrPrev) equals false, no operation is executed.) *)
	END_VAR

END_FUNCTION

// Functions/Geometric and Coordinate Transformations/F_VN_ApplyScalingToAffineTransformation

	{attribute 'TcIecLibraryType'}
	{attribute 'external_name' := 'F_VN_ApplyScalingToAffineTransformation_GUID_71143E90_5D49_54DF_44FC_B90F2833E712'}
	(* Apply a scaling to an existing 2D affine transformation matrix. *)
	FUNCTION F_VN_ApplyScalingToAffineTransformation : HRESULT
	VAR_INPUT
		aTransformationMatrix	:	REFERENCE TO TcVnMatrix2x3_LREAL;	(* Affine transformation matrix to which the scaling is applied *)
		fScaleX	:	LREAL;	(* Scaling factor in x direction *)
		fScaleY	:	LREAL;	(* Scaling factor in y direction *)
		hrPrev	:	HRESULT;	(* HRESULT indicating the result of previous operations (If SUCCEEDED(hrPrev) equals false, no operation is executed.) *)
	END_VAR

END_FUNCTION

// Functions/Geometric and Coordinate Transformations/F_VN_ApplyScalingToAffineTransformationExp

	{attribute 'TcIecLibraryType'}
	{attribute 'external_name' := 'F_VN_ApplyScalingToAffineTransformationExp_GUID_70CA841F_34F9_5F8F_792E_E49DCD592CBB'}
	(* Apply a scaling to an existing 2D affine transformation matrix. (expert function) *)
	FUNCTION F_VN_ApplyScalingToAffineTransformationExp : HRESULT
	VAR_INPUT
		aTransformationMatrix	:	REFERENCE TO TcVnMatrix2x3_LREAL;	(* Affine transformation matrix to which the scaling is applied *)
		fScaleX	:	LREAL;	(* Scaling factor in x direction *)
		fScaleY	:	LREAL;	(* Scaling factor in y direction *)
		bUsePreMultiplication	:	BOOL;	(* Select if pre- or post-multiplication should be used *)
		hrPrev	:	HRESULT;	(* HRESULT indicating the result of previous operations (If SUCCEEDED(hrPrev) equals false, no operation is executed.) *)
	END_VAR

END_FUNCTION

// Functions/Geometric and Coordinate Transformations/F_VN_ApplyTranslationToAffineTransformation

	{attribute 'TcIecLibraryType'}
	{attribute 'external_name' := 'F_VN_ApplyTranslationToAffineTransformation_GUID_57347F47_DB22_5AAF_4003_1498E26B983A'}
	(* Apply a translation to an existing 2D affine transformation matrix. *)
	FUNCTION F_VN_ApplyTranslationToAffineTransformation : HRESULT
	VAR_INPUT
		aTransformationMatrix	:	REFERENCE TO TcVnMatrix2x3_LREAL;	(* Affine transformation matrix to which the translation is applied *)
		fDeltaX	:	LREAL;	(* Translation in x direction *)
		fDeltaY	:	LREAL;	(* Translation in y direction *)
		hrPrev	:	HRESULT;	(* HRESULT indicating the result of previous operations (If SUCCEEDED(hrPrev) equals false, no operation is executed.) *)
	END_VAR

END_FUNCTION

// Functions/Geometric and Coordinate Transformations/F_VN_ApplyTranslationToAffineTransformationExp

	{attribute 'TcIecLibraryType'}
	{attribute 'external_name' := 'F_VN_ApplyTranslationToAffineTransformationExp_GUID_CF594AFD_ABA4_5183_4850_4C8999CAB10F'}
	(* Apply a translation to an existing 2D affine transformation matrix. (expert function) *)
	FUNCTION F_VN_ApplyTranslationToAffineTransformationExp : HRESULT
	VAR_INPUT
		aTransformationMatrix	:	REFERENCE TO TcVnMatrix2x3_LREAL;	(* Affine transformation matrix to which the translation is applied *)
		fDeltaX	:	LREAL;	(* Translation in x direction *)
		fDeltaY	:	LREAL;	(* Translation in y direction *)
		bUsePreMultiplication	:	BOOL;	(* Select if pre- or post-multiplication should be used *)
		hrPrev	:	HRESULT;	(* HRESULT indicating the result of previous operations (If SUCCEEDED(hrPrev) equals false, no operation is executed.) *)
	END_VAR

END_FUNCTION

// Functions/Geometric and Coordinate Transformations/F_VN_ApplyYAxisInversionToAffineTransformation

	{attribute 'TcIecLibraryType'}
	{attribute 'external_name' := 'F_VN_ApplyYAxisInversionToAffineTransformation_GUID_D070F0B3_5A51_5231_762F_B47FE2915795'}
	(* Apply an inversion of the y-axis direction to an existing 2D affine transformation matrix. *)
	FUNCTION F_VN_ApplyYAxisInversionToAffineTransformation : HRESULT
	VAR_INPUT
		aTransformationMatrix	:	REFERENCE TO TcVnMatrix2x3_LREAL;	(* Affine transformation matrix to which the inversion of the y-axis direction is applied *)
		hrPrev	:	HRESULT;	(* HRESULT indicating the result of previous operations (If SUCCEEDED(hrPrev) equals false, no operation is executed.) *)
	END_VAR

END_FUNCTION

// Functions/Geometric and Coordinate Transformations/F_VN_ApplyYAxisInversionToAffineTransformationExp

	{attribute 'TcIecLibraryType'}
	{attribute 'external_name' := 'F_VN_ApplyYAxisInversionToAffineTransformationExp_GUID_7ECE7C1D_7BB2_5FDB_5015_44B90C76F392'}
	(* Apply an inversion of the y-axis direction to an existing 2D affine transformation matrix. (expert function) *)
	FUNCTION F_VN_ApplyYAxisInversionToAffineTransformationExp : HRESULT
	VAR_INPUT
		aTransformationMatrix	:	REFERENCE TO TcVnMatrix2x3_LREAL;	(* Affine transformation matrix to which the inversion of the y-axis direction is applied *)
		bUsePreMultiplication	:	BOOL;	(* Select if pre- or post-multiplication should be used *)
		hrPrev	:	HRESULT;	(* HRESULT indicating the result of previous operations (If SUCCEEDED(hrPrev) equals false, no operation is executed.) *)
	END_VAR

END_FUNCTION

// Functions/Geometric and Coordinate Transformations/F_VN_ConvertCartesianToPolarAngleImage

